# B&R Automation Studio project NAEUL004C00R13L518F00 (part 28)

#### Act_OptP1040Save.st
```iecst
ACTION Act_OptP1040Save:

	IF tyP1040ProdSet.tyProdSet.tyBtnSave.bRtCompl = TRUE THEN
		IF usiSaveProdRcpStep = 0 THEN
			//Mask Table
			tyP1040ProdSet.tyProdSet.tyStringSearch.uiMaskRtStat				:= FALSE;
			tyP1040ProdSet.tyProdSet.tyTableRecipe.uiMaskRtStat					:= FALSE;
			tyP1040ProdSet.tyProdSet.tyBtnDelete.uiMaskRtStat					:= FALSE;

			p_tyC0008MsgBox ACCESS ADR(tyP1040ProdSet.tyMsgBoxSaveAsk);

			IF tyP1040ProdSet.tyMsgBoxSaveAsk.tyBtnYes.bRtCompl = TRUE THEN
				tyP1040ProdSet.tyMsgBoxSaveAsk.tyBtnYes.bRtCompl				:= FALSE;
				tyP1040ProdSet.tyMsgBoxSaveAsk.tyBtnYes.bValue					:= FALSE;

				p_tyC0008MsgBox ACCESS ADR(tyP1040ProdSet.tyMsgBoxHide);

				usiSaveProdRcpStep	:= 1;

			ELSIF tyP1040ProdSet.tyMsgBoxSaveAsk.tyBtnNo.bRtCompl = TRUE THEN
				tyP1040ProdSet.tyMsgBoxSaveAsk.tyBtnNo.bRtCompl					:= FALSE;
				tyP1040ProdSet.tyMsgBoxSaveAsk.tyBtnNo.bValue					:= FALSE;

				p_tyC0008MsgBox ACCESS ADR(tyP1040ProdSet.tyMsgBoxHide);

				usiSaveProdRcpStep	:= 99;

			END_IF

		ELSIF usiSaveProdRcpStep = 1 THEN
			tyProdRcpInfoIn.sRcpNm				:= tyP1040ProdSet.tyProdSet.tyStringRecipeNm.sValue;
			tyProdRcpInfoIn.diWidthInUM			:= tyP1040ProdSet.tyProdSet.tyNumProdWidth.diValue;
			tyProdRcpInfoIn.diMaxSltValue		:= tyP1040ProdSet.tyProdSet.tyNumLastSlt.diValue;
			tyProdRcpInfoIn.diMinSltValue		:= tyP1040ProdSet.tyProdSet.tyNumFirstSlt.diValue;
			tyProdRcpInfoIn.diPitch				:= tyP1040ProdSet.tyProdSet.tyNumPitch.diValue;
			tyProdRcpInfoIn.diBrdPerSlt			:= tyP1040ProdSet.tyProdSet.tyNumBrdPerSlt.diValue;
			tyProdRcpInfoIn.usiMcMod			:= tyP1040ProdSet.tyProdSet.tyDrpDnMcMode.usiValueIdx;
			tyProdRcpInfoIn.bTopToBtm			:= tyP1040ProdSet.tyProdSet.tyBtnToptoBtm.bValue;
			tyProdRcpInfoIn.bGapBwtnBrd			:= tyP1040ProdSet.tyProdSet.tyBtnGapBetBrds.bValue;
			tyProdRcpInfoIn.bLongBrd			:= tyP1040ProdSet.tyProdSet.tyBtnLongBrd.bValue;
			tyProdRcpInfoIn.diMinReqFreeBffr	:= tyP1040ProdSet.tyProdSet.tyNumMinReqFreeBffr.diValue;
			tyProdRcpInfoIn.diMtrPshrExtSpd		:= tyP1040ProdSet.tyProdSet.tyNumMtrPshrExtSpd.diValue;
			tyProdRcpInfoIn.diMtrPshrExtTorq	:= tyP1040ProdSet.tyProdSet.tyNumMtrPshrExtTorq.diValue;
			tyProdRcpInfoIn.diPshrOffset		:= tyP1040ProdSet.tyProdSet.tyNumPshrOffset.diValue;

			IF p_tyNtParamCurr.bLFProdWidth2Prep THEN
				tyProdRcpInfoIn.diWidthInUM2		:= tyP1040ProdSet.tyProdSet.tyNumProdWidth2.diValue;// ADD
			ELSE
				tyProdRcpInfoIn.diWidthInUM2		:= tyP1040ProdSet.tyProdSet.tyNumProdWidth.diValue;// ADD
			END_IF

			eProdRcpAct	:= ProdRcpActAddEdit;

			IF p_eProdRcpStat = ProdRcpActAddEdit AND p_eProdRcpStatus = Done THEN
				eProdRcpAct	:= ProdRcpActIdle;

				IF p_bProdRcpNmEmpty = TRUE THEN
					usiSaveProdRcpStep		:= 2;
				ELSIF p_bProdRcpListFull = TRUE THEN
					usiSaveProdRcpStep		:= 3;
				ELSE
					tyP1040ProdSet.tyProdSet.tyBtnSort.bValue := FALSE;
					bRefreshProdRcpTable	:= TRUE;
					bRefreshProdRcpDetail	:= TRUE;
					usiSaveProdRcpStep		:= 4;
				END_IF

			ELSIF p_eProdRcpStatus = Error THEN
				p_tyC0008MsgBox ACCESS ADR(tyP1040ProdSet.tyMsgBoxSaveErr);

				IF tyP1040ProdSet.tyMsgBoxSaveErr.tyBtnNo.bRtCompl = TRUE THEN
					tyP1040ProdSet.tyMsgBoxSaveErr.tyBtnNo.bRtCompl 			:= FALSE;
					tyP1040ProdSet.tyMsgBoxSaveErr.tyBtnNo.bValue 				:= FALSE;

					p_tyC0008MsgBox ACCESS ADR(tyP1040ProdSet.tyMsgBoxHide);

					usiSaveProdRcpStep		:= 99;
				END_IF
			END_IF

		// Product Recipe Param Error
		ELSIF usiSaveProdRcpStep = 2 THEN
			p_tyC0008MsgBox ACCESS ADR(tyP1040ProdSet.tyMsgBoxSaveNoNm);

			IF tyP1040ProdSet.tyMsgBoxSaveNoNm.tyBtnNo.bRtCompl = TRUE THEN
				tyP1040ProdSet.tyMsgBoxSaveNoNm.tyBtnNo.bRtCompl 				:= FALSE;
				tyP1040ProdSet.tyMsgBoxSaveNoNm.tyBtnNo.bValue 					:= FALSE;

				p_tyC0008MsgBox ACCESS ADR(tyP1040ProdSet.tyMsgBoxHide);

				usiSaveProdRcpStep		:= 99;
			END_IF

		// Prod Recipe List Full
		ELSIF usiSaveProdRcpStep = 3 THEN
			p_tyC0008MsgBox ACCESS ADR(tyP1040ProdSet.tyMsgBoxListFull);

			IF tyP1040ProdSet.tyMsgBoxListFull.tyBtnNo.bRtCompl = TRUE THEN
				tyP1040ProdSet.tyMsgBoxListFull.tyBtnNo.bRtCompl 				:= FALSE;
				tyP1040ProdSet.tyMsgBoxListFull.tyBtnNo.bValue 					:= FALSE;

				p_tyC0008MsgBox ACCESS ADR(tyP1040ProdSet.tyMsgBoxHide);

				usiSaveProdRcpStep		:= 99;
			END_IF

		ELSIF usiSaveProdRcpStep = 4 THEN
			IF tyProdRcpInfoIn.sRcpNm = p_tyProdRcpCurrRcp0.sRcpNm THEN
				p_tyC0008MsgBox ACCESS ADR(tyP1040ProdSet.tyMsgBoxReloadCurrRcp);

				IF tyP1040ProdSet.tyMsgBoxReloadCurrRcp.tyBtnNo.bRtCompl = TRUE THEN
					tyP1040ProdSet.tyMsgBoxReloadCurrRcp.tyBtnNo.bRtCompl 		:= FALSE;
					tyP1040ProdSet.tyMsgBoxReloadCurrRcp.tyBtnNo.bValue 		:= FALSE;

					p_tyC0008MsgBox ACCESS ADR(tyP1040ProdSet.tyMsgBoxHide);

					usiSaveProdRcpStep		:= 99;
				END_IF
			ELSE
				usiSaveProdRcpStep			:= 99;
			END_IF

		ELSIF usiSaveProdRcpStep = 99 THEN
			bRefreshProdRcpTable 			:= FALSE;

			//Unmask
			tyP1040ProdSet.tyProdSet.tyStringSearch.uiMaskRtStat	:= TRUE;
			tyP1040ProdSet.tyProdSet.tyTableRecipe.uiMaskRtStat		:= TRUE;
			tyP1040ProdSet.tyProdSet.tyBtnDelete.uiMaskRtStat		:= TRUE;

			//Reset
			tyP1040ProdSet.tyProdSet.tyBtnSave.bRtCompl	:= FALSE;
			tyP1040ProdSet.tyProdSet.tyBtnSave.bValue	:= FALSE;

			usiSaveProdRcpStep	:= 0;

		END_IF

	END_IF

END_ACTION
```

#### Act_OptP1040LoadData.st
```iecst
ACTION Act_OptP1040LoadData:

	udiP1040SelectedRow		:= STRING_TO_UDINT(tyP1040ProdSet.tyProdSet.tyTableRecipe.a_tyStringDataCol0[tyP1040Table.uiSelectedRow].sValue);

	IF udiP1040SelectedRow <> udiP1040SelectedRowOld OR bRefreshProdRcpDetail = TRUE OR bUpdateP1040LoadData THEN
		IF tyP1040ProdSet.tyProdSet.tyStringSearch.sValue = '' THEN
			IF tyP1040ProdSet.tyProdSet.tyTableRecipe.a_tyStringDataCol1[tyP1040Table.uiSelectedRow].sValue <> '' THEN
				//Update Recipe Data
				IF tyP1040ProdSet.tyProdSet.tyBtnSort.bValue THEN
					tyP1040ProdSet.tyProdSet.tyStringRecipeNm.sValue		:= p_tyProdRcpSortedList[udiP1040SelectedRow].sRcpNm;
					tyP1040ProdSet.tyProdSet.tyNumProdWidth.diValue			:= p_tyProdRcpSortedList[udiP1040SelectedRow].diWidthInUM;
					tyP1040ProdSet.tyProdSet.tyNumProdWidth2.diValue		:= p_tyProdRcpSortedList[udiP1040SelectedRow].diWidthInUM2;
					tyP1040ProdSet.tyProdSet.tyNumLastSlt.diValue			:= p_tyProdRcpSortedList[udiP1040SelectedRow].diMaxSltValue;
					tyP1040ProdSet.tyProdSet.tyNumFirstSlt.diValue			:= p_tyProdRcpSortedList[udiP1040SelectedRow].diMinSltValue;
					tyP1040ProdSet.tyProdSet.tyNumPitch.diValue				:= p_tyProdRcpSortedList[udiP1040SelectedRow].diPitch;
					tyP1040ProdSet.tyProdSet.tyNumBrdPerSlt.diValue			:= p_tyProdRcpSortedList[udiP1040SelectedRow].diBrdPerSlt;
					tyP1040ProdSet.tyProdSet.tyDrpDnMcMode.usiValueIdx		:= p_tyProdRcpSortedList[udiP1040SelectedRow].usiMcMod;
					tyP1040ProdSet.tyProdSet.tyBtnToptoBtm.bValue			:= p_tyProdRcpSortedList[udiP1040SelectedRow].bTopToBtm;
					tyP1040ProdSet.tyProdSet.tyBtnGapBetBrds.bValue			:= p_tyProdRcpSortedList[udiP1040SelectedRow].bGapBwtnBrd;
					tyP1040ProdSet.tyProdSet.tyBtnLongBrd.bValue			:= p_tyProdRcpSortedList[udiP1040SelectedRow].bLongBrd;
					tyP1040ProdSet.tyProdSet.tyNumMinReqFreeBffr.diValue	:= p_tyProdRcpSortedList[udiP1040SelectedRow].diMinReqFreeBffr;
					tyP1040ProdSet.tyProdSet.tyNumMtrPshrExtSpd.diValue		:= p_tyProdRcpSortedList[udiP1040SelectedRow].diMtrPshrExtSpd;
					tyP1040ProdSet.tyProdSet.tyNumMtrPshrExtTorq.diValue	:= p_tyProdRcpSortedList[udiP1040SelectedRow].diMtrPshrExtTorq;
					tyP1040ProdSet.tyProdSet.tyNumPshrOffset.diValue		:= p_tyProdRcpSortedList[udiP1040SelectedRow].diPshrOffset;
				ELSE

					tyP1040ProdSet.tyProdSet.tyStringRecipeNm.sValue		:= p_tyProdRcpCurrList[udiP1040SelectedRow].sRcpNm;
					tyP1040ProdSet.tyProdSet.tyNumProdWidth.diValue			:= p_tyProdRcpCurrList[udiP1040SelectedRow].diWidthInUM;
					tyP1040ProdSet.tyProdSet.tyNumProdWidth2.diValue		:= p_tyProdRcpCurrList[udiP1040SelectedRow].diWidthInUM2;
					tyP1040ProdSet.tyProdSet.tyNumLastSlt.diValue			:= p_tyProdRcpCurrList[udiP1040SelectedRow].diMaxSltValue;
					tyP1040ProdSet.tyProdSet.tyNumFirstSlt.diValue			:= p_tyProdRcpCurrList[udiP1040SelectedRow].diMinSltValue;
					tyP1040ProdSet.tyProdSet.tyNumPitch.diValue				:= p_tyProdRcpCurrList[udiP1040SelectedRow].diPitch;
					tyP1040ProdSet.tyProdSet.tyNumBrdPerSlt.diValue			:= p_tyProdRcpCurrList[udiP1040SelectedRow].diBrdPerSlt;
					tyP1040ProdSet.tyProdSet.tyDrpDnMcMode.usiValueIdx		:= p_tyProdRcpCurrList[udiP1040SelectedRow].usiMcMod;
					tyP1040ProdSet.tyProdSet.tyBtnToptoBtm.bValue			:= p_tyProdRcpCurrList[udiP1040SelectedRow].bTopToBtm;
					tyP1040ProdSet.tyProdSet.tyBtnGapBetBrds.bValue			:= p_tyProdRcpCurrList[udiP1040SelectedRow].bGapBwtnBrd;
					tyP1040ProdSet.tyProdSet.tyBtnLongBrd.bValue			:= p_tyProdRcpCurrList[udiP1040SelectedRow].bLongBrd;
					tyP1040ProdSet.tyProdSet.tyNumMinReqFreeBffr.diValue	:= p_tyProdRcpCurrList[udiP1040SelectedRow].diMinReqFreeBffr;
					tyP1040ProdSet.tyProdSet.tyNumMtrPshrExtSpd.diValue		:= p_tyProdRcpCurrList[udiP1040SelectedRow].diMtrPshrExtSpd;
					tyP1040ProdSet.tyProdSet.tyNumMtrPshrExtTorq.diValue	:= p_tyProdRcpCurrList[udiP1040SelectedRow].diMtrPshrExtTorq;
					tyP1040ProdSet.tyProdSet.tyNumPshrOffset.diValue		:= p_tyProdRcpCurrList[udiP1040SelectedRow].diPshrOffset;
				END_IF
			ELSE
				tyP1040ProdSet.tyProdSet.tyStringRecipeNm.sValue		:= '';
				tyP1040ProdSet.tyProdSet.tyNumProdWidth.diValue			:= 100000;
				tyP1040ProdSet.tyProdSet.tyNumProdWidth2.diValue		:= 100000;
				tyP1040ProdSet.tyProdSet.tyNumLastSlt.diValue			:= p_tyMagRcpCurrRcp.diTtlSlt;
				tyP1040ProdSet.tyProdSet.tyNumFirstSlt.diValue			:= p_tyNtParamCurr.diProjMagMinSlt;
				tyP1040ProdSet.tyProdSet.tyNumPitch.diValue				:= 1;
				tyP1040ProdSet.tyProdSet.tyNumBrdPerSlt.diValue			:= 1;
				tyP1040ProdSet.tyProdSet.tyDrpDnMcMode.usiValueIdx		:= p_tyMcParamCurr.usiDefaultMcMod;
				tyP1040ProdSet.tyProdSet.tyBtnToptoBtm.bValue			:= FALSE;
				tyP1040ProdSet.tyProdSet.tyBtnGapBetBrds.bValue			:= FALSE;
				tyP1040ProdSet.tyProdSet.tyBtnLongBrd.bValue			:= FALSE;
				tyP1040ProdSet.tyProdSet.tyNumMinReqFreeBffr.diValue	:= 0;
				tyP1040ProdSet.tyProdSet.tyNumMtrPshrExtSpd.diValue		:= 8;
				tyP1040ProdSet.tyProdSet.tyNumMtrPshrExtTorq.diValue	:= 80;
				tyP1040ProdSet.tyProdSet.tyNumPshrOffset.diValue		:= 0;
			END_IF

		ELSE

			IF tyP1040ProdSet.tyProdSet.tyTableRecipe.a_tyStringDataCol1[tyP1040Table.uiSelectedRow].sValue <> '' THEN
				//Update Recipe Data
				IF tyP1040ProdSet.tyProdSet.tyBtnSort.bValue THEN
					tyP1040ProdSet.tyProdSet.tyStringRecipeNm.sValue		:= p_tyProdRcpSortedList[udiP1040SelectedRow].sRcpNm;
					tyP1040ProdSet.tyProdSet.tyNumProdWidth.diValue			:= p_tyProdRcpSortedList[udiP1040SelectedRow].diWidthInUM;
					tyP1040ProdSet.tyProdSet.tyNumProdWidth2.diValue		:= p_tyProdRcpSortedList[udiP1040SelectedRow].diWidthInUM2;
					tyP1040ProdSet.tyProdSet.tyNumLastSlt.diValue			:= p_tyProdRcpSortedList[udiP1040SelectedRow].diMaxSltValue;
					tyP1040ProdSet.tyProdSet.tyNumFirstSlt.diValue			:= p_tyProdRcpSortedList[udiP1040SelectedRow].diMinSltValue;
					tyP1040ProdSet.tyProdSet.tyNumPitch.diValue				:= p_tyProdRcpSortedList[udiP1040SelectedRow].diPitch;
					tyP1040ProdSet.tyProdSet.tyNumBrdPerSlt.diValue			:= p_tyProdRcpSortedList[udiP1040SelectedRow].diBrdPerSlt;
					tyP1040ProdSet.tyProdSet.tyDrpDnMcMode.usiValueIdx		:= p_tyProdRcpSortedList[udiP1040SelectedRow].usiMcMod;
					tyP1040ProdSet.tyProdSet.tyBtnToptoBtm.bValue			:= p_tyProdRcpSortedList[udiP1040SelectedRow].bTopToBtm;
					tyP1040ProdSet.tyProdSet.tyBtnGapBetBrds.bValue			:= p_tyProdRcpSortedList[udiP1040SelectedRow].bGapBwtnBrd;
					tyP1040ProdSet.tyProdSet.tyBtnLongBrd.bValue			:= p_tyProdRcpSortedList[udiP1040SelectedRow].bLongBrd;
					tyP1040ProdSet.tyProdSet.tyNumMinReqFreeBffr.diValue	:= p_tyProdRcpSortedList[udiP1040SelectedRow].diMinReqFreeBffr;
					tyP1040ProdSet.tyProdSet.tyNumMtrPshrExtSpd.diValue		:= p_tyProdRcpSortedList[udiP1040SelectedRow].diMtrPshrExtSpd;
					tyP1040ProdSet.tyProdSet.tyNumMtrPshrExtTorq.diValue	:= p_tyProdRcpSortedList[udiP1040SelectedRow].diMtrPshrExtTorq;
					tyP1040ProdSet.tyProdSet.tyNumPshrOffset.diValue		:= p_tyProdRcpSortedList[udiP1040SelectedRow].diPshrOffset;
				ELSE
					tyP1040ProdSet.tyProdSet.tyStringRecipeNm.sValue		:= p_tyProdRcpFilterList[udiP1040SelectedRow].sRcpNm;
					tyP1040ProdSet.tyProdSet.tyNumProdWidth.diValue			:= p_tyProdRcpFilterList[udiP1040SelectedRow].diWidthInUM;
					tyP1040ProdSet.tyProdSet.tyNumProdWidth2.diValue		:= p_tyProdRcpSortedList[udiP1040SelectedRow].diWidthInUM2;
					tyP1040ProdSet.tyProdSet.tyNumLastSlt.diValue			:= p_tyProdRcpFilterList[udiP1040SelectedRow].diMaxSltValue;
					tyP1040ProdSet.tyProdSet.tyNumFirstSlt.diValue			:= p_tyProdRcpFilterList[udiP1040SelectedRow].diMinSltValue;
					tyP1040ProdSet.tyProdSet.tyNumPitch.diValue				:= p_tyProdRcpFilterList[udiP1040SelectedRow].diPitch;
					tyP1040ProdSet.tyProdSet.tyNumBrdPerSlt.diValue			:= p_tyProdRcpFilterList[udiP1040SelectedRow].diBrdPerSlt;
					tyP1040ProdSet.tyProdSet.tyDrpDnMcMode.usiValueIdx		:= p_tyProdRcpFilterList[udiP1040SelectedRow].usiMcMod;
					tyP1040ProdSet.tyProdSet.tyBtnToptoBtm.bValue			:= p_tyProdRcpFilterList[udiP1040SelectedRow].bTopToBtm;
					tyP1040ProdSet.tyProdSet.tyBtnGapBetBrds.bValue			:= p_tyProdRcpFilterList[udiP1040SelectedRow].bGapBwtnBrd;
					tyP1040ProdSet.tyProdSet.tyBtnLongBrd.bValue			:= p_tyProdRcpFilterList[udiP1040SelectedRow].bLongBrd;
					tyP1040ProdSet.tyProdSet.tyNumMinReqFreeBffr.diValue	:= p_tyProdRcpFilterList[udiP1040SelectedRow].diMinReqFreeBffr;
					tyP1040ProdSet.tyProdSet.tyNumMtrPshrExtSpd.diValue		:= p_tyProdRcpFilterList[udiP1040SelectedRow].diMtrPshrExtSpd;
					tyP1040ProdSet.tyProdSet.tyNumMtrPshrExtTorq.diValue	:= p_tyProdRcpFilterList[udiP1040SelectedRow].diMtrPshrExtTorq;
					tyP1040ProdSet.tyProdSet.tyNumPshrOffset.diValue		:= p_tyProdRcpFilterList[udiP1040SelectedRow].diPshrOffset;
				END_IF
			ELSE
				tyP1040ProdSet.tyProdSet.tyStringRecipeNm.sValue		:= '';
				tyP1040ProdSet.tyProdSet.tyNumProdWidth.diValue			:= 100000;
				tyP1040ProdSet.tyProdSet.tyNumProdWidth2.diValue		:= 100000;
				tyP1040ProdSet.tyProdSet.tyNumLastSlt.diValue			:= p_tyMagRcpCurrRcp.diTtlSlt;
				tyP1040ProdSet.tyProdSet.tyNumFirstSlt.diValue			:= p_tyNtParamCurr.diProjMagMinSlt;
				tyP1040ProdSet.tyProdSet.tyNumPitch.diValue				:= 1;
				tyP1040ProdSet.tyProdSet.tyNumBrdPerSlt.diValue			:= 1;
				tyP1040ProdSet.tyProdSet.tyDrpDnMcMode.usiValueIdx		:= p_tyMcParamCurr.usiDefaultMcMod;
				tyP1040ProdSet.tyProdSet.tyBtnToptoBtm.bValue			:= FALSE;
				tyP1040ProdSet.tyProdSet.tyBtnGapBetBrds.bValue			:= FALSE;
				tyP1040ProdSet.tyProdSet.tyBtnLongBrd.bValue			:= FALSE;
				tyP1040ProdSet.tyProdSet.tyNumMinReqFreeBffr.diValue	:= 0;
				tyP1040ProdSet.tyProdSet.tyNumMtrPshrExtSpd.diValue		:= 8;
				tyP1040ProdSet.tyProdSet.tyNumMtrPshrExtTorq.diValue	:= 80;
				tyP1040ProdSet.tyProdSet.tyNumPshrOffset.diValue		:= 0;
			END_IF

		END_IF

		bUpdateP1040LoadData 		:= FALSE;
		bRefreshProdRcpDetail		:= FALSE;
		udiP1040SelectedRowOld 		:= udiP1040SelectedRow;

		fUIInRtStatOff(ADR(tyP1040ProdSet.tyProdSet.tyBtnSave.uiMaskRtStat));

	END_IF

END_ACTION
```

#### Act_OptP1040Del.st
```iecst
ACTION Act_OptP1040Del:

	IF tyP1040ProdSet.tyProdSet.tyBtnDelete.bRtCompl = TRUE THEN
		IF usiDelProdRcpStep = 0 THEN
			tyP1040ProdSet.tyProdSet.tyStringSearch.uiMaskRtStat				:= FALSE;
			tyP1040ProdSet.tyProdSet.tyTableRecipe.uiMaskRtStat					:= FALSE;

			IF tyP1040ProdSet.tyProdSet.tyTableRecipe.a_tyStringDataCol1[tyP1040Table.uiSelectedRow].sValue = p_tyProdRcpCurrRcp0.sRcpNm THEN
				p_tyC0008MsgBox ACCESS ADR(tyP1040ProdSet.tyMsgBoxDelCurrRcpAsk);

				IF tyP1040ProdSet.tyMsgBoxDelCurrRcpAsk.tyBtnNo.bRtCompl = TRUE THEN
					tyP1040ProdSet.tyMsgBoxDelCurrRcpAsk.tyBtnNo.bRtCompl 		:= FALSE;
					tyP1040ProdSet.tyMsgBoxDelCurrRcpAsk.tyBtnNo.bValue 		:= FALSE;

					p_tyC0008MsgBox ACCESS ADR(tyP1040ProdSet.tyMsgBoxHide);

					usiDelProdRcpStep	:= 99;
				END_IF
			ELSE
				p_tyC0008MsgBox ACCESS ADR(tyP1040ProdSet.tyMsgBoxDelAsk);

				IF tyP1040ProdSet.tyMsgBoxDelAsk.tyBtnYes.bRtCompl = TRUE THEN
					tyP1040ProdSet.tyMsgBoxDelAsk.tyBtnYes.bRtCompl				:= FALSE;
					tyP1040ProdSet.tyMsgBoxDelAsk.tyBtnYes.bValue				:= FALSE;

					p_tyC0008MsgBox ACCESS ADR(tyP1040ProdSet.tyMsgBoxHide);

					usiDelProdRcpStep	:= 1;

				ELSIF tyP1040ProdSet.tyMsgBoxDelAsk.tyBtnNo.bRtCompl = TRUE THEN
					tyP1040ProdSet.tyMsgBoxDelAsk.tyBtnNo.bRtCompl				:= FALSE;
					tyP1040ProdSet.tyMsgBoxDelAsk.tyBtnNo.bValue				:= FALSE;

					p_tyC0008MsgBox ACCESS ADR(tyP1040ProdSet.tyMsgBoxHide);

					usiDelProdRcpStep	:= 99;

				END_IF
			END_IF

		ELSIF usiDelProdRcpStep = 1 THEN
			tyProdRcpInfoIn.sRcpNm			:= tyP1040ProdSet.tyProdSet.tyTableRecipe.a_tyStringDataCol1[tyP1040Table.uiSelectedRow].sValue;

			eProdRcpAct					:= ProdRcpActDel;

			IF p_eProdRcpStat = ProdRcpActDel AND p_eProdRcpStatus = Done THEN
				eProdRcpAct				:= ProdRcpActIdle;

				IF p_bProdRcpNmEmpty = TRUE THEN
					usiDelProdRcpStep		:= 2;
				ELSIF p_bProdRcpNmNotExist = TRUE THEN
					usiDelProdRcpStep		:= 3;
				ELSE
					tyP1040ProdSet.tyProdSet.tyBtnSort.bValue := FALSE;
					bRefreshProdRcpTable	:= TRUE;
					bRefreshProdRcpDetail	:= TRUE;
					usiDelProdRcpStep		:= 99;
				END_IF

			ELSIF p_eProdRcpStatus = Error THEN
				p_tyC0008MsgBox ACCESS ADR(tyP1040ProdSet.tyMsgBoxDelErr);

				IF tyP1040ProdSet.tyMsgBoxDelErr.tyBtnNo.bRtCompl = TRUE THEN
					tyP1040ProdSet.tyMsgBoxDelErr.tyBtnNo.bRtCompl 				:= FALSE;
					tyP1040ProdSet.tyMsgBoxDelErr.tyBtnNo.bValue 				:= FALSE;

					p_tyC0008MsgBox ACCESS ADR(tyP1040ProdSet.tyMsgBoxHide);

					usiDelProdRcpStep		:= 99;
				END_IF
			END_IF

		ELSIF usiDelProdRcpStep = 2 THEN
			p_tyC0008MsgBox ACCESS ADR(tyP1040ProdSet.tyMsgBoxDelNmEmpty);

			IF tyP1040ProdSet.tyMsgBoxDelNmEmpty.tyBtnNo.bRtCompl = TRUE THEN
				tyP1040ProdSet.tyMsgBoxDelNmEmpty.tyBtnNo.bRtCompl 				:= FALSE;
				tyP1040ProdSet.tyMsgBoxDelNmEmpty.tyBtnNo.bValue 				:= FALSE;

				p_tyC0008MsgBox ACCESS ADR(tyP1040ProdSet.tyMsgBoxHide);

				usiDelProdRcpStep		:= 99;
			END_IF

		ELSIF usiDelProdRcpStep = 3 THEN
			p_tyC0008MsgBox ACCESS ADR(tyP1040ProdSet.tyMsgBoxDelNmNotExist);

			IF tyP1040ProdSet.tyMsgBoxDelNmNotExist.tyBtnNo.bRtCompl = TRUE THEN
				tyP1040ProdSet.tyMsgBoxDelNmNotExist.tyBtnNo.bRtCompl 		:= FALSE;
				tyP1040ProdSet.tyMsgBoxDelNmNotExist.tyBtnNo.bValue 		:= FALSE;

				p_tyC0008MsgBox ACCESS ADR(tyP1040ProdSet.tyMsgBoxHide);

				usiDelProdRcpStep	:= 99;
			END_IF

		ELSIF usiDelProdRcpStep = 99 THEN
			bRefreshProdRcpTable	:= FALSE;

			//Unmask
			tyP1040ProdSet.tyProdSet.tyStringSearch.uiMaskRtStat			:= TRUE;
			tyP1040ProdSet.tyProdSet.tyTableRecipe.uiMaskRtStat				:= TRUE;

			//Reset
			tyP1040ProdSet.tyProdSet.tyBtnDelete.bRtCompl					:= FALSE;
			tyP1040ProdSet.tyProdSet.tyBtnDelete.bValue						:= FALSE;

			usiDelProdRcpStep		:= 0;
		END_IF

	END_IF

END_ACTION
```

#### Act_OptP1040Table.st
```iecst
ACTION Act_OptP1040Table:

	//Call Table FB
	fbP1040Table.sVisuNm			:= tyP1040Table.sVisuNm;
	fbP1040Table.udiWorkAreaStartX	:= 359;
	fbP1040Table.udiWorkAreaEndX	:= 770;
	fbP1040Table.udiWorkAreaStartY	:= 93;
	fbP1040Table.udiWorkAreaEndY	:= 415;
	fbP1040Table.udiMinXDist		:= 20;
	fbP1040Table.udiMinYDist		:= 20;
	fbP1040Table.uiSlideScale		:= c_uiP1040TableSize;
	fbP1040Table.iTotalData			:= UDINT_TO_INT(c_udiProdRcpMax);
	fbP1040Table.iTotalRow			:= c_uiP1040TableSize;
	fbP1040Table.p_uiSliderStatus	:= ADR(tyP1040ProdSet.tyProdSet.tyTableRecipe.tyUISlider.uiRtStat);
	fbP1040Table.pa_tyUIHotspot		:= ADR(tyP1040ProdSet.tyProdSet.tyTableRecipe.a_tyHotspot);
	fbP1040Table.p_uiTablePos		:= ADR(tyP1040Table.uiTablePos);
	fbP1040Table.p_iSliderPos		:= ADR(tyP1040ProdSet.tyProdSet.tyTableRecipe.tyUISlider.iValue);
	fbP1040Table.p_uiSelectedRow	:= ADR(tyP1040Table.uiSelectedRow);
	fbP1040Table.p_bTableActive		:= ADR(tyP1040Table.bTableActive);
	fbP1040Table.p_bSliderActive	:= ADR(tyP1040Table.bSliderActive);
	fbP1040Table;

	//Table Content
	IF tyP1040Table.bTableActive = TRUE OR tyP1040Table.bSliderActive = TRUE OR bRefreshProdRcpTable = TRUE OR bUpdateP1040Table THEN
		FOR i := 1 TO c_uiP1040TableSize DO
			IF tyP1040ProdSet.tyProdSet.tyBtnSort.bValue THEN
				tyP1040ProdSet.tyProdSet.tyTableRecipe.a_tyStringDataCol0[i].sValue	    := UINT_TO_STRING(tyP1040Table.uiTablePos + i - 1);
				tyP1040ProdSet.tyProdSet.tyTableRecipe.a_tyStringDataCol1[i].sValue		:= p_tyProdRcpSortedList[tyP1040Table.uiTablePos + i - 1].sRcpNm;
				tyP1040ProdSet.tyProdSet.tyTableRecipe.a_tyStringDataCol2[i].sValue		:= p_tyProdRcpSortedList[tyP1040Table.uiTablePos + i - 1].sDisplayInfo;
			ELSE

				IF tyP1040ProdSet.tyProdSet.tyStringSearch.sValue = '' THEN
					tyP1040ProdSet.tyProdSet.tyTableRecipe.a_tyStringDataCol0[i].sValue	    := UINT_TO_STRING(tyP1040Table.uiTablePos + i - 1);
					tyP1040ProdSet.tyProdSet.tyTableRecipe.a_tyStringDataCol1[i].sValue		:= p_tyProdRcpCurrList[tyP1040Table.uiTablePos + i - 1].sRcpNm;
					tyP1040ProdSet.tyProdSet.tyTableRecipe.a_tyStringDataCol2[i].sValue		:= p_tyProdRcpCurrList[tyP1040Table.uiTablePos + i - 1].sDisplayInfo;
				ELSE
					tyP1040ProdSet.tyProdSet.tyTableRecipe.a_tyStringDataCol0[i].sValue		:= UINT_TO_STRING(tyP1040Table.uiTablePos + i - 1);
					tyP1040ProdSet.tyProdSet.tyTableRecipe.a_tyStringDataCol1[i].sValue		:= p_tyProdRcpFilterList[tyP1040Table.uiTablePos + i - 1].sRcpNm;
					tyP1040ProdSet.tyProdSet.tyTableRecipe.a_tyStringDataCol2[i].sValue		:= p_tyProdRcpFilterList[tyP1040Table.uiTablePos + i - 1].sDisplayInfo;
				END_IF
			END_IF

		END_FOR

		IF bUpdateP1040Table THEN
			bUpdateP1040Table := FALSE;
		END_IF
	END_IF

	//Selected Row
	IF tyP1040Table.uiSelectedRow <> tyP1040Table.uiSelectedRowOld THEN
		FOR i := 1 TO c_uiP1040TableSize DO
			IF tyP1040Table.uiSelectedRow = i THEN
				tyP1040ProdSet.tyProdSet.tyTableRecipe.a_tyStringDataCol1[i].usiColor	:= 1;
				tyP1040ProdSet.tyProdSet.tyTableRecipe.a_tyStringDataCol2[i].usiColor	:= 1;
			ELSE
				tyP1040ProdSet.tyProdSet.tyTableRecipe.a_tyStringDataCol1[i].usiColor	:= 0;
				tyP1040ProdSet.tyProdSet.tyTableRecipe.a_tyStringDataCol2[i].usiColor	:= 0;
			END_IF
		END_FOR

		tyP1040Table.uiSelectedRowOld	:= tyP1040Table.uiSelectedRow;
	END_IF

END_ACTION
```

#### Act_OptP1040Search.st
```iecst
ACTION Act_OptP1040Search:

	IF tyP1040ProdSet.tyProdSet.tyStringSearch.bRtCompl = TRUE THEN	//Search Input Valid
		IF tyP1040ProdSet.tyProdSet.tyStringSearch.sValue = '' THEN
			FOR i := 1 TO c_uiP1040TableSize DO
				tyP1040ProdSet.tyProdSet.tyTableRecipe.a_tyStringDataCol0[i].sValue			:= UINT_TO_STRING(tyP1040Table.uiTablePos + i - 1);
				tyP1040ProdSet.tyProdSet.tyTableRecipe.a_tyStringDataCol1[i].sValue			:= p_tyProdRcpCurrList[tyP1040Table.uiTablePos + i - 1].sRcpNm;
				tyP1040ProdSet.tyProdSet.tyTableRecipe.a_tyStringDataCol2[i].sValue			:= p_tyProdRcpCurrList[tyP1040Table.uiTablePos + i - 1].sDisplayInfo;
			END_FOR

			tyP1040ProdSet.tyProdSet.tyStringSearch.bRtCompl			:= FALSE;
			bRefreshProdRcpDetail										:= TRUE;

			IF tyP1040ProdSet.tyProdSet.tyBtnSort.bValue THEN
				bFilterSortP1040	:= TRUE;
			END_IF

		ELSE
			tyP1040ProdSet.tyProdSet.tyTableRecipe.uiMaskRtStat			:= FALSE;
			tyP1040ProdSet.tyProdSet.tyBtnSave.uiMaskRtStat				:= FALSE;
			tyP1040ProdSet.tyProdSet.tyBtnDelete.uiMaskRtStat			:= FALSE;

			sProdRcpSearch			:= tyP1040ProdSet.tyProdSet.tyStringSearch.sValue;

			eProdRcpAct			:= ProdRcpActFilter;

			IF p_eProdRcpStat = ProdRcpActFilter AND p_eProdRcpStatus = Done THEN
				eProdRcpAct		:= ProdRcpActIdle;

				FOR i := 1 TO c_uiP1040TableSize DO
					tyP1040ProdSet.tyProdSet.tyTableRecipe.a_tyStringDataCol0[i].sValue		:= UINT_TO_STRING(tyP1040Table.uiTablePos + i - 1);
					tyP1040ProdSet.tyProdSet.tyTableRecipe.a_tyStringDataCol1[i].sValue		:= p_tyProdRcpFilterList[tyP1040Table.uiTablePos + i - 1].sRcpNm;
					tyP1040ProdSet.tyProdSet.tyTableRecipe.a_tyStringDataCol2[i].sValue		:= p_tyProdRcpFilterList[tyP1040Table.uiTablePos + i - 1].sDisplayInfo;
				END_FOR

				//Unmask Table
				tyP1040ProdSet.tyProdSet.tyTableRecipe.uiMaskRtStat		:= TRUE;
				tyP1040ProdSet.tyProdSet.tyBtnSave.uiMaskRtStat			:= FALSE;
				tyP1040ProdSet.tyProdSet.tyBtnDelete.uiMaskRtStat		:= TRUE;

				//Reset
				tyP1040ProdSet.tyProdSet.tyStringSearch.bRtCompl		:= FALSE;
				bRefreshProdRcpDetail									:= TRUE;

				IF tyP1040ProdSet.tyProdSet.tyBtnSort.bValue THEN
					bFilterSortP1040	:= TRUE;
				END_IF

			ELSIF p_eProdRcpStatus = Error THEN
				FOR i := 1 TO c_uiP1040TableSize DO
					tyP1040ProdSet.tyProdSet.tyTableRecipe.a_tyStringDataCol0[i].sValue		:= UINT_TO_STRING(tyP1040Table.uiTablePos + i - 1);
					tyP1040ProdSet.tyProdSet.tyTableRecipe.a_tyStringDataCol1[i].sValue		:= '';
					tyP1040ProdSet.tyProdSet.tyTableRecipe.a_tyStringDataCol2[i].sValue		:= '';
				END_FOR

				p_tyC0008MsgBox ACCESS ADR (tyP1040ProdSet.tyMsgBoxListErr);

				IF tyP1040ProdSet.tyMsgBoxListErr.tyBtnNo.bRtCompl = TRUE THEN
					tyP1040ProdSet.tyMsgBoxListErr.tyBtnNo.bRtCompl 	:= TRUE;
					tyP1040ProdSet.tyMsgBoxListErr.tyBtnNo.bValue		:= TRUE;

					p_tyC0008MsgBox ACCESS ADR (tyP1040ProdSet.tyMsgBoxHide);

					//Unmask Table
					tyP1040ProdSet.tyProdSet.tyTableRecipe.uiMaskRtStat	:= TRUE;
					tyP1040ProdSet.tyProdSet.tyBtnSave.uiMaskRtStat		:= FALSE;
					tyP1040ProdSet.tyProdSet.tyBtnDelete.uiMaskRtStat	:= TRUE;

					//Reset
					tyP1040ProdSet.tyProdSet.tyStringSearch.bRtCompl	:= FALSE;
					bRefreshProdRcpDetail								:= TRUE;
				END_IF
			END_IF
		END_IF
	END_IF

END_ACTION
```

#### Act_OptP1040Keypad.st
```iecst
ACTION Act_OptP1040Keypad:

	tyP1040ProdSet.tyProdSet.tyNumFirstSlt.diValueMax	:= tyP1040ProdSet.tyProdSet.tyNumLastSlt.diValue;
	tyP1040ProdSet.tyProdSet.tyNumLastSlt.diValueMin	:= tyP1040ProdSet.tyProdSet.tyNumFirstSlt.diValue;
	tyP1040ProdSet.tyProdSet.tyNumPitch.diValueMax		:= tyP1040ProdSet.tyProdSet.tyNumLastSlt.diValue - tyP1040ProdSet.tyProdSet.tyNumFirstSlt.diValue + 1;

	IF fUIOutRtStatTPIsOpen(ADR(tyP1040ProdSet.tyProdSet.tyStringRecipeNm.uiRtStat)) THEN
		tyProperty.tyKeypad.tyStringTitle.sKeypadTitle	:= tyP1040ProdSet.tyProdSet.tyStringRecipeNm.sKeypadTitle;

	ELSIF fUIOutRtStatTPIsOpen(ADR(tyP1040ProdSet.tyProdSet.tyNumProdWidth.uiRtStat)) THEN
		IF p_tyNtParamCurr.bLFProdWidth2Prep THEN
			tyProperty.tyKeypad.tyTxtTitle.sTxt	:= 'Product Width US';
		ELSE
			tyProperty.tyKeypad.tyTxtTitle.sTxt	:= 'Product Width';
		END_IF

	ELSIF fUIOutRtStatTPIsOpen(ADR(tyP1040ProdSet.tyProdSet.tyNumProdWidth2.uiRtStat)) THEN
		tyProperty.tyKeypad.tyTxtTitle.sTxt	:='Product Width DS';

	ELSIF fUIOutRtStatTPIsOpen(ADR(tyP1040ProdSet.tyProdSet.tyStringSearch.uiRtStat)) THEN
		tyProperty.tyKeypad.tyStringTitle.sKeypadTitle	:= tyP1040ProdSet.tyProdSet.tyStringSearch.sKeypadTitle;

	ELSIF fUIOutRtStatTPIsOpen(ADR(tyP1040ProdSet.tyProdSet.tyNumFirstSlt.uiRtStat)) THEN
		tyProperty.tyKeypad.tyStringTitle.sKeypadTitle	:= tyP1040ProdSet.tyProdSet.tyNumFirstSlt.sKeypadTitle;

	ELSIF fUIOutRtStatTPIsOpen(ADR(tyP1040ProdSet.tyProdSet.tyNumLastSlt.uiRtStat)) THEN
		tyProperty.tyKeypad.tyStringTitle.sKeypadTitle	:= tyP1040ProdSet.tyProdSet.tyNumLastSlt.sKeypadTitle;

	ELSIF fUIOutRtStatTPIsOpen(ADR(tyP1040ProdSet.tyProdSet.tyNumPitch.uiRtStat)) THEN
		tyProperty.tyKeypad.tyStringTitle.sKeypadTitle	:= tyP1040ProdSet.tyProdSet.tyNumPitch.sKeypadTitle;

	ELSIF fUIOutRtStatTPIsOpen(ADR(tyP1040ProdSet.tyProdSet.tyNumMinReqFreeBffr.uiRtStat)) THEN
		tyProperty.tyKeypad.tyStringTitle.sKeypadTitle	:= tyP1040ProdSet.tyProdSet.tyNumMinReqFreeBffr.sKeypadTitle;

	ELSIF fUIOutRtStatTPIsOpen(ADR(tyP1040ProdSet.tyProdSet.tyNumBrdPerSlt.uiRtStat)) THEN
		tyProperty.tyKeypad.tyStringTitle.sKeypadTitle	:= tyP1040ProdSet.tyProdSet.tyNumBrdPerSlt.sKeypadTitle;

	ELSIF fUIOutRtStatTPIsOpen(ADR(tyP1040ProdSet.tyProdSet.tyNumPshrOffset.uiRtStat))THEN
		tyProperty.tyKeypad.tyStringTitle.sKeypadTitle	:= tyP1040ProdSet.tyProdSet.tyNumPshrOffset.sKeypadTitle;

	ELSE
		tyProperty.tyKeypad.tyStringTitle.sKeypadTitle	:= '';

	END_IF

END_ACTION
```

#### Act_OptP1040Limit.st
```iecst
ACTION Act_OptP1040Limit:

//	IF tyP1040ProdSet.tyProdSet.tyTableRecipe.a_tyStringDataCol1[udiP1040SelectedRow].sValue <> '' THEN
//		tyP1040ProdSet.tyProdSet.tyNumPshrOffset.diValueMin		:= -(p_tyProdRcpCurrList[udiP1040SelectedRow].diWidthInUM/2-p_tyMcParamCurr.diAWPusherAtHmPosInUM-5000);
//		tyP1040ProdSet.tyProdSet.tyNumPshrOffset.diValueMax		:= (p_tyProdRcpCurrList[udiP1040SelectedRow].diWidthInUM/2-p_tyMcParamCurr.diAWPusherAtHmPosInUM-5000);
//	ELSE
//		tyP1040ProdSet.tyProdSet.tyNumPshrOffset.diValueMin		:= 0;
//		tyP1040ProdSet.tyProdSet.tyNumPshrOffset.diValueMax		:= 0;
//	END_IF

	//Pusher Offset has to include min safe zone and max safe zone for the product width // 04102022 - 2022-0617
	IF (tyP1040ProdSet.tyProdSet.tyNumProdWidth.diValue) <> 0 THEN
		tyP1040ProdSet.tyProdSet.tyNumPshrOffset.diValueMin	:= - ((tyP1040ProdSet.tyProdSet.tyNumProdWidth.diValue/2 - p_tyMcParamCurr.diAWPusherAtHmPosInUM) - IPshrSafeDistanceValue);
		tyP1040ProdSet.tyProdSet.tyNumPshrOffset.diValueMax	:= ((tyP1040ProdSet.tyProdSet.tyNumProdWidth.diValue/2 - p_tyMcParamCurr.diAWPusherAtHmPosInUM) - IPshrSafeDistanceValue);
	ELSE
		tyP1040ProdSet.tyProdSet.tyNumPshrOffset.diValueMin	:= 0;
		tyP1040ProdSet.tyProdSet.tyNumPshrOffset.diValueMax	:= 0;
	END_IF

END_ACTION
```

#### Act_OptP1040Sort.st
```iecst
ACTION Act_OptP1040Sort:

	IF tyP1040ProdSet.tyProdSet.tyBtnSort.bValue THEN
		tyP1040ProdSet.tyProdSet.tyBtnSort.usiTxtIdx 	:= 1;
	ELSE
		tyP1040ProdSet.tyProdSet.tyBtnSort.usiTxtIdx 	:= 0;
	END_IF

	IF tyP1040ProdSet.tyProdSet.tyBtnSort.bRtCompl THEN
		bUpdateP1040LoadData := TRUE;
	END_IF

	IF tyP1040ProdSet.tyProdSet.tyBtnSort.bRtCompl OR (bFilterSortP1040 AND p_eProdRcpStat<> ProdRcpActFilter) THEN

		IF tyP1040ProdSet.tyProdSet.tyBtnSort.bValue THEN

			tyP1040ProdSet.tyProdSet.tyTableRecipe.uiMaskRtStat.0	:= FALSE;

			sProdRcpSearch	:= tyP1040ProdSet.tyProdSet.tyStringSearch.sValue;

			eProdRcpAct	:= ProdRcpActSort;

			IF p_eProdRcpStat = ProdRcpActSort AND p_eProdRcpStatus = Done THEN
				eProdRcpAct		:= ProdRcpActIdle;

				FOR i := 1 TO c_uiP1040TableSize DO
					tyP1040ProdSet.tyProdSet.tyTableRecipe.a_tyStringDataCol0[i].sValue	:= UINT_TO_STRING(tyP1040Table.uiTablePos + i - 1);
					tyP1040ProdSet.tyProdSet.tyTableRecipe.a_tyStringDataCol1[i].sValue	:= p_tyProdRcpSortedList[tyP1040Table.uiTablePos + i - 1].sRcpNm;
					tyP1040ProdSet.tyProdSet.tyTableRecipe.a_tyStringDataCol2[i].sValue	:= p_tyProdRcpSortedList[tyP1040Table.uiTablePos + i - 1].sDisplayInfo;
				END_FOR

				bFilterSortP1040	:= FALSE;

				//Unmask
				tyP1040ProdSet.tyProdSet.tyTableRecipe.uiMaskRtStat.0	:= TRUE;

				tyP1040ProdSet.tyProdSet.tyBtnSort.bRtCompl := FALSE;

			ELSIF p_eProdRcpStatus = Error THEN
				FOR i := 1 TO c_uiP1040TableSize DO
					tyP1040ProdSet.tyProdSet.tyTableRecipe.a_tyStringDataCol0[i].sValue		:= UINT_TO_STRING(tyP1040Table.uiTablePos + i - 1);
					tyP1040ProdSet.tyProdSet.tyTableRecipe.a_tyStringDataCol1[i].sValue		:= '';
					tyP1040ProdSet.tyProdSet.tyTableRecipe.a_tyStringDataCol2[i].sValue		:= '';
				END_FOR

				p_tyC0008MsgBox ACCESS ADR (tyP1040ProdSet.tyMsgBoxListErr);

				bFilterSortP1040	:= FALSE;

				IF tyP1040ProdSet.tyMsgBoxListErr.tyBtnNo.bRtCompl = TRUE THEN
					tyP1040ProdSet.tyMsgBoxListErr.tyBtnNo.bRtCompl 		:= TRUE;
					tyP1040ProdSet.tyMsgBoxListErr.tyBtnNo.bValue			:= TRUE;

					p_tyC0008MsgBox ACCESS ADR (tyP1040ProdSet.tyMsgBoxHide);

					//Unmask
					tyP1040ProdSet.tyProdSet.tyTableRecipe.uiMaskRtStat.0	:= TRUE;

					//Reset
					tyP1040ProdSet.tyProdSet.tyBtnSort.bRtCompl := FALSE;
				END_IF
			END_IF

		ELSE

			bUpdateP1040Table	:= TRUE;

			tyP1040ProdSet.tyProdSet.tyBtnSort.bRtCompl := FALSE;

		END_IF

	END_IF

END_ACTION
```

#### Act_OptP1040ToXML.st
```iecst
ACTION Act_OptP1040ToXML:

	IF tyP1040ProdSet.tyProdSet.tyBtnToXML.bRtCompl = TRUE THEN

		IF usiProdRcpToXMLStep = 0 THEN
			//Confirmation Message - To XML Ask
			//Mask
			fUIInRtStatOff(ADR(tyP1040ProdSet.tyProdSet.tyStringSearch.uiMaskRtStat));
			fUIInRtStatOff(ADR(tyP1040ProdSet.tyProdSet.tyTableRecipe.uiMaskRtStat));

			p_tyC0008MsgBox ACCESS ADR(tyP1040ProdSet.tyMsgBoxToXMLAsk);

			IF tyP1040ProdSet.tyMsgBoxToXMLAsk.tyBtnYes.bRtCompl = TRUE THEN
				tyP1040ProdSet.tyMsgBoxToXMLAsk.tyBtnYes.bRtCompl	:= FALSE;
				tyP1040ProdSet.tyMsgBoxToXMLAsk.tyBtnYes.bValue		:= FALSE;

				p_tyC0008MsgBox ACCESS ADR(tyP1040ProdSet.tyMsgBoxHide);

				usiProdRcpToXMLStep	:= 1;

			ELSIF tyP1040ProdSet.tyMsgBoxToXMLAsk.tyBtnNo.bRtCompl = TRUE THEN
				tyP1040ProdSet.tyMsgBoxToXMLAsk.tyBtnNo.bRtCompl	:= FALSE;
				tyP1040ProdSet.tyMsgBoxToXMLAsk.tyBtnNo.bValue		:= FALSE;

				p_tyC0008MsgBox ACCESS ADR(tyP1040ProdSet.tyMsgBoxHide);

				usiProdRcpToXMLStep	:= 99;
			END_IF

		ELSIF usiProdRcpToXMLStep = 1 THEN
			//Save Recipe To XML
			eMpProdRcpAct	:= MpProdRcpActSave;

			IF p_eMpProdRcpStat = MpProdRcpActSave AND p_eMpProdRcpStatus = Done THEN
				eMpProdRcpAct	:= MpProdRcpActIdle;

				tyP1040ProdSet.tyProdSet.tyBtnSort.bValue := FALSE;
				bRefreshProdRcpTable	:= TRUE;
				bRefreshProdRcpDetail	:= TRUE;

				usiProdRcpToXMLStep		:= 99;

			ELSIF p_eMpProdRcpStatus = Error THEN
				p_tyC0008MsgBox ACCESS ADR(tyP1040ProdSet.tyMsgBoxToXMLErr);

				IF tyP1040ProdSet.tyMsgBoxToXMLErr.tyBtnNo.bRtCompl = TRUE THEN
					tyP1040ProdSet.tyMsgBoxToXMLErr.tyBtnNo.bRtCompl	:= FALSE;
					tyP1040ProdSet.tyMsgBoxToXMLErr.tyBtnNo.bValue		:= FALSE;

					p_tyC0008MsgBox ACCESS ADR(tyP1040ProdSet.tyMsgBoxHide);

					usiProdRcpToXMLStep	:= 99;
				END_IF

			END_IF

		ELSIF usiProdRcpToXMLStep = 99 THEN
			//Complete Reset
			bRefreshProdRcpTable	:= FALSE;

			//Unmask
			fUIInRtStatHide(ADR(tyP1040ProdSet.tyProdSet.tyStringSearch.uiMaskRtStat));
			fUIInRtStatHide(ADR(tyP1040ProdSet.tyProdSet.tyTableRecipe.uiMaskRtStat));

			tyP1040ProdSet.tyProdSet.tyBtnToXML.bRtCompl	:= FALSE;
			tyP1040ProdSet.tyProdSet.tyBtnToXML.bValue		:= FALSE;

			usiProdRcpToXMLStep	:= 0;

		END_IF

	END_IF

END_ACTION
```

#### Act_OptP1040FromXML.st
```iecst
ACTION Act_OptP1040FromXML:

	IF tyP1040ProdSet.tyProdSet.tyBtnFromXML.bRtCompl = TRUE THEN

		IF usiProdRcpFromXMLStep = 0 THEN
			//Confirmation Message - From XML Ask
			//Mask
			fUIInRtStatOff(ADR(tyP1040ProdSet.tyProdSet.tyStringSearch.uiMaskRtStat));
			fUIInRtStatOff(ADR(tyP1040ProdSet.tyProdSet.tyTableRecipe.uiMaskRtStat));

			p_tyC0008MsgBox ACCESS ADR(tyP1040ProdSet.tyMsgBoxFromXMLAsk);

			IF tyP1040ProdSet.tyMsgBoxFromXMLAsk.tyBtnYes.bRtCompl = TRUE THEN
				tyP1040ProdSet.tyMsgBoxFromXMLAsk.tyBtnYes.bRtCompl	:= FALSE;
				tyP1040ProdSet.tyMsgBoxFromXMLAsk.tyBtnYes.bValue	:= FALSE;

				p_tyC0008MsgBox ACCESS ADR(tyP1040ProdSet.tyMsgBoxHide);

				usiProdRcpFromXMLStep	:= 1;

			ELSIF tyP1040ProdSet.tyMsgBoxFromXMLAsk.tyBtnNo.bRtCompl = TRUE THEN
				tyP1040ProdSet.tyMsgBoxFromXMLAsk.tyBtnNo.bRtCompl	:= FALSE;
				tyP1040ProdSet.tyMsgBoxFromXMLAsk.tyBtnNo.bValue	:= FALSE;

				p_tyC0008MsgBox ACCESS ADR(tyP1040ProdSet.tyMsgBoxHide);

				usiProdRcpFromXMLStep	:= 99;
			END_IF

		ELSIF usiProdRcpFromXMLStep = 1 THEN
			//Load Recipe From XML
			eMpProdRcpAct	:= MpProdRcpActLoad;

			IF p_eMpProdRcpStat = MpProdRcpActLoad AND p_eMpProdRcpStatus = Done THEN
				eMpProdRcpAct	:= MpProdRcpActIdle;

				tyP1040ProdSet.tyProdSet.tyBtnSort.bValue      := FALSE;
				tyP1040ProdSet.tyProdSet.tyStringSearch.sValue := '';
				bRefreshProdRcpTable	:= TRUE;
				bRefreshProdRcpDetail	:= TRUE;

				usiProdRcpFromXMLStep	:= 2;

			ELSIF p_eMpProdRcpStatus = Error THEN
				p_tyC0008MsgBox ACCESS ADR(tyP1040ProdSet.tyMsgBoxFromXMLErr);

				IF tyP1040ProdSet.tyMsgBoxFromXMLErr.tyBtnNo.bRtCompl = TRUE THEN
					tyP1040ProdSet.tyMsgBoxFromXMLErr.tyBtnNo.bRtCompl	:= FALSE;
					tyP1040ProdSet.tyMsgBoxFromXMLErr.tyBtnNo.bValue	:= FALSE;

					p_tyC0008MsgBox ACCESS ADR(tyP1040ProdSet.tyMsgBoxHide);

					usiProdRcpFromXMLStep	:= 99;
				END_IF

			END_IF

		ELSIF usiProdRcpFromXMLStep = 2 THEN
			//Save Product Recipe List
			eProdRcpAct	:= ProdRcpActSaveList;

			IF p_eProdRcpStat = ProdRcpActSaveList AND p_eProdRcpStatus = Done THEN
				eProdRcpAct	:= ProdRcpActIdle;

				usiProdRcpFromXMLStep	:= 99;

			ELSIF p_eProdRcpStatus = Error THEN
				p_tyC0008MsgBox ACCESS ADR(tyP1040ProdSet.tyMsgBoxSaveListErr);

				IF tyP1040ProdSet.tyMsgBoxSaveListErr.tyBtnNo.bRtCompl = TRUE THEN
					tyP1040ProdSet.tyMsgBoxSaveListErr.tyBtnNo.bRtCompl	:= FALSE;
					tyP1040ProdSet.tyMsgBoxSaveListErr.tyBtnNo.bValue	:= FALSE;

					p_tyC0008MsgBox ACCESS ADR(tyP1040ProdSet.tyMsgBoxHide);

					usiProdRcpFromXMLStep	:= 99;
				END_IF

			END_IF

		ELSIF usiProdRcpFromXMLStep = 99 THEN
			//Complete Reset
			bRefreshProdRcpTable	:= FALSE;

			//Unmask
			fUIInRtStatHide(ADR(tyP1040ProdSet.tyProdSet.tyStringSearch.uiMaskRtStat));
			fUIInRtStatHide(ADR(tyP1040ProdSet.tyProdSet.tyTableRecipe.uiMaskRtStat));

			tyP1040ProdSet.tyProdSet.tyBtnFromXML.bRtCompl	:= FALSE;
			tyP1040ProdSet.tyProdSet.tyBtnFromXML.bValue	:= FALSE;

			usiProdRcpFromXMLStep	:= 0;

		END_IF

	END_IF

END_ACTION
```

#### Act_EntP1050Disp.st
```iecst
ACTION Act_EntP1050Disp:

	//Access Address
	p_tyC0005Main ACCESS ADR(tyCommon.tyMain);

	p_tyC0006Set ACCESS ADR(tyCommon.tySet);

	p_tyC0007Notif ACCESS ADR(tyCommon.tyNotif);

	p_tyC0008MsgBox ACCESS ADR(tyP1050LFSet.tyMsgBoxHide);

	p_tyC0009Info ACCESS ADR(tyCommon.tyInfo);

	p_tyP1050LFSetLdrEdit ACCESS ADR(tyP1050LFSet.tyLdrEdit);
	p_tyP1050LFSetLdr ACCESS ADR(tyP1050LFSet.tyLdr);

END_ACTION
```

#### Act_OptP1050Edit.st
```iecst
ACTION Act_OptP1050Edit:

	IF tyP1050LFSet.tyLdr.tyBtnEdit.bRtCompl = TRUE THEN

		FOR i := 1 TO UDINT_TO_UINT(c_diLFClntNum) DO
			IF tyMcParamWr.a_sLFIPAddr[i] = '' THEN
				uiLFStartEditNo	:= i;
				EXIT;
			END_IF
		END_FOR

		tyP1050LFSet.tyLdr.tyBtnEdit.bRtCompl	:= FALSE;
		tyP1050LFSet.tyLdr.tyBtnEdit.bValue		:= TRUE;

		fUIInRtStatOff(ADR(tyP1050LFSet.tyLdrEdit.tyLyr.uiRtStat));
		fUIInRtStatHide(ADR(tyP1050LFSet.tyLdr.tyLyr.uiRtStat));

		tyP1050LFSet.tyLdrEdit.tyNumMcNum.diValue		:= STRING_TO_DINT(tyP1050LFSet.tyLdr.tyTable1List.a_tyStringDataCol0[tyP1050Table.uiSelectedRow].sValue);
		tyP1050LFSet.tyLdrEdit.tyStringIPAddr.sValue	:= tyP1050LFSet.tyLdr.tyTable1List.a_tyStringDataCol2[tyP1050Table.uiSelectedRow].sValue;

	ELSIF tyP1050LFSet.tyLdr.tyBtnEdit.bValue = TRUE THEN

		IF tyP1050LFSet.tyLdrEdit.tyBtnOk.bRtCompl = TRUE THEN

			IF fIPValid(tyP1050LFSet.tyLdrEdit.tyStringIPAddr.sValue , ADR(a_iIPPart1)) = TRUE AND bCheckDone = FALSE THEN
				FOR i := 1 TO UDINT_TO_UINT(c_diLFClntNum) DO
					IF i <>  tyP1050Table.uiTablePos + tyP1050Table.uiSelectedRow - 1 THEN
						fIPValid(p_tyMcParamCurr.a_sLFIPAddr[i] , ADR(a_iIPPart2));

						IF (a_iIPPart1[1] = a_iIPPart2[1] AND a_iIPPart1[2] = a_iIPPart2[2] AND a_iIPPart1[3] = a_iIPPart2[3] AND a_iIPPart1[4] = a_iIPPart2[4])
							AND (tyP1050LFSet.tyLdrEdit.tyStringIPAddr.sValue <> '') THEN

							bIPDuplicate	:= TRUE;
							EXIT;

						END_IF
					END_IF
				END_FOR
				bCheckDone := TRUE;
			END_IF

			IF fIPValid(tyP1050LFSet.tyLdrEdit.tyStringIPAddr.sValue , ADR(a_iIPPart1)) = FALSE THEN
				p_tyC0008MsgBox ACCESS ADR(tyP1050LFSet.tyMsgBoxIPAddrInvalid);

				IF tyP1050LFSet.tyMsgBoxIPAddrInvalid.tyBtnNo.bRtCompl = TRUE THEN
					tyP1050LFSet.tyMsgBoxIPAddrInvalid.tyBtnNo.bRtCompl	:= FALSE;
					tyP1050LFSet.tyMsgBoxIPAddrInvalid.tyBtnNo.bValue	:= FALSE;

					p_tyC0008MsgBox ACCESS ADR(tyP1050LFSet.tyMsgBoxHide);

					tyP1050LFSet.tyLdrEdit.tyBtnOk.bRtCompl	:= FALSE;
					tyP1050LFSet.tyLdrEdit.tyBtnOk.bValue	:= FALSE;
					bCheckDone := FALSE;
				END_IF

			ELSIF bIPDuplicate = TRUE THEN
				p_tyC0008MsgBox ACCESS ADR(tyP1050LFSet.tyMsgBoxIPAddrDuplicate);

				IF tyP1050LFSet.tyMsgBoxIPAddrDuplicate.tyBtnNo.bRtCompl = TRUE THEN
					tyP1050LFSet.tyMsgBoxIPAddrDuplicate.tyBtnNo.bRtCompl	:= FALSE;
					tyP1050LFSet.tyMsgBoxIPAddrDuplicate.tyBtnNo.bValue		:= FALSE;

					p_tyC0008MsgBox ACCESS ADR(tyP1050LFSet.tyMsgBoxHide);

					bIPDuplicate							:= FALSE;
					tyP1050LFSet.tyLdrEdit.tyBtnOk.bRtCompl	:= FALSE;
					tyP1050LFSet.tyLdrEdit.tyBtnOk.bValue	:= FALSE;
					bCheckDone := FALSE;
				END_IF
			ELSE
				IF tyP1050LFSet.tyLdr.tyTable1List.a_tyStringDataCol2[tyP1050Table.uiSelectedRow].sValue = '' THEN
					tyMcParamWr.a_sLFIPAddr[uiLFStartEditNo]	:= tyP1050LFSet.tyLdrEdit.tyStringIPAddr.sValue;

					eMcParamAct	:= McParamActWrite;

					IF p_eMcParamStat = McParamActWrite AND p_eMcParamStatus = Done THEN
						eMcParamAct	:= McParamActIdle;

						tyP1050LFSet.tyLdr.tyTable1List.a_tyStringDataCol2[uiLFStartEditNo].sValue		:= tyP1050LFSet.tyLdrEdit.tyStringIPAddr.sValue;

						IF tyP1050LFSet.tyLdrEdit.tyStringIPAddr.sValue = '0000' THEN
							tyP1050LFSet.tyLdr.tyTable1List.a_tyTxtDataCol3[uiLFStartEditNo].usiValueIdx	:= 3;
						ELSE
							tyP1050LFSet.tyLdr.tyTable1List.a_tyTxtDataCol3[uiLFStartEditNo].usiValueIdx	:= 1;
						END_IF

						//LF Control
						FOR i := 1 TO c_uiP1050TableSize DO
							tyP0700LFCtrl.tyLdr.tyTable1List.a_tyStringDataCol0[i].sValue	:= UINT_TO_STRING(tyP0700Table.uiTablePos + i - 1);
							tyP0700LFCtrl.tyLdr.tyTable1List.a_tyStringDataCol2[i].sValue	:= p_tyMcParamCurr.a_sLFIPAddr[tyP0700Table.uiTablePos + i - 1];
						END_FOR

						tyP1050LFSet.tyLdrEdit.tyBtnOk.bRtCompl	:= FALSE;
						tyP1050LFSet.tyLdrEdit.tyBtnOk.bValue	:= FALSE;
						tyP1050LFSet.tyLdr.tyBtnEdit.bValue		:= FALSE;
						bCheckDone								:= FALSE;

						bUpdateP1050Table	:=TRUE;

						fUIInRtStatHide(ADR(tyP1050LFSet.tyLdrEdit.tyLyr.uiRtStat));
						fUIInRtStatOff(ADR(tyP1050LFSet.tyLdr.tyLyr.uiRtStat));

					ELSIF p_eMcParamStatus = Error THEN
						p_tyC0008MsgBox ACCESS ADR(tyP1050LFSet.tyMsgBoxSaveErr);

						IF tyP1050LFSet.tyMsgBoxSaveErr.tyBtnNo.bRtCompl = TRUE THEN
							tyP1050LFSet.tyMsgBoxSaveErr.tyBtnNo.bRtCompl	:= FALSE;
							tyP1050LFSet.tyMsgBoxSaveErr.tyBtnNo.bValue		:= FALSE;

							p_tyC0008MsgBox ACCESS ADR(tyP1050LFSet.tyMsgBoxHide);

							//Recover
							tyMcParamWr	:= p_tyMcParamCurr;

							tyP1050LFSet.tyLdrEdit.tyBtnOk.bRtCompl	:= FALSE;
							tyP1050LFSet.tyLdrEdit.tyBtnOk.bValue	:= FALSE;
							tyP1050LFSet.tyLdr.tyBtnEdit.bValue		:= FALSE;
							bCheckDone								:=FALSE;

							fUIInRtStatHide(ADR(tyP1050LFSet.tyLdrEdit.tyLyr.uiRtStat));
							fUIInRtStatOff(ADR(tyP1050LFSet.tyLdr.tyLyr.uiRtStat));
						END_IF
					END_IF
				ELSE
					tyMcParamWr.a_sLFIPAddr[tyP1050Table.uiTablePos + tyP1050Table.uiSelectedRow - 1]	:= tyP1050LFSet.tyLdrEdit.tyStringIPAddr.sValue;

					eMcParamAct	:= McParamActWrite;

					IF p_eMcParamStat = McParamActWrite AND p_eMcParamStatus = Done THEN
						eMcParamAct	:= McParamActIdle;

						tyP1050LFSet.tyLdr.tyTable1List.a_tyStringDataCol2[tyP1050Table.uiSelectedRow].sValue		:= tyP1050LFSet.tyLdrEdit.tyStringIPAddr.sValue;

						IF tyP1050LFSet.tyLdrEdit.tyStringIPAddr.sValue = '0000' THEN
							tyP1050LFSet.tyLdr.tyTable1List.a_tyTxtDataCol3[tyP1050Table.uiSelectedRow].usiValueIdx	:= 3;
						ELSE
							tyP1050LFSet.tyLdr.tyTable1List.a_tyTxtDataCol3[ tyP1050Table.uiSelectedRow].usiValueIdx	:= 1;
						END_IF

						//LF Control
						FOR i := 1 TO c_uiP1050TableSize DO
							tyP0700LFCtrl.tyLdr.tyTable1List.a_tyStringDataCol0[i].sValue	:= UINT_TO_STRING(tyP0700Table.uiTablePos + i - 1);
							tyP0700LFCtrl.tyLdr.tyTable1List.a_tyStringDataCol2[i].sValue	:= p_tyMcParamCurr.a_sLFIPAddr[tyP0700Table.uiTablePos + i - 1];
						END_FOR

						tyP1050LFSet.tyLdrEdit.tyBtnOk.bRtCompl	:= FALSE;
						tyP1050LFSet.tyLdrEdit.tyBtnOk.bValue	:= FALSE;
						tyP1050LFSet.tyLdr.tyBtnEdit.bValue		:= FALSE;
						bCheckDone								:= FALSE;

						fUIInRtStatHide(ADR(tyP1050LFSet.tyLdrEdit.tyLyr.uiRtStat));
						fUIInRtStatOff(ADR(tyP1050LFSet.tyLdr.tyLyr.uiRtStat));

					ELSIF p_eMcParamStatus = Error THEN

						p_tyC0008MsgBox ACCESS ADR(tyP1050LFSet.tyMsgBoxSaveErr);

						IF tyP1050LFSet.tyMsgBoxSaveErr.tyBtnNo.bRtCompl = TRUE THEN
							tyP1050LFSet.tyMsgBoxSaveErr.tyBtnNo.bRtCompl	:= FALSE;
							tyP1050LFSet.tyMsgBoxSaveErr.tyBtnNo.bValue		:= FALSE;

							p_tyC0008MsgBox ACCESS ADR(tyP1050LFSet.tyMsgBoxHide);

							//Recover
							tyMcParamWr	:= p_tyMcParamCurr;

							tyP1050LFSet.tyLdrEdit.tyBtnOk.bRtCompl	:= FALSE;
							tyP1050LFSet.tyLdrEdit.tyBtnOk.bValue	:= FALSE;
							tyP1050LFSet.tyLdr.tyBtnEdit.bValue		:= FALSE;
							bCheckDone								:=FALSE;

							fUIInRtStatHide(ADR(tyP1050LFSet.tyLdrEdit.tyLyr.uiRtStat));
							fUIInRtStatOff(ADR(tyP1050LFSet.tyLdr.tyLyr.uiRtStat));
						END_IF
					END_IF
				END_IF
			END_IF

		ELSIF tyP1050LFSet.tyLdrEdit.tyBtnCancel.bRtCompl = TRUE THEN
			tyP1050LFSet.tyLdrEdit.tyBtnCancel.bRtCompl	:= FALSE;
			tyP1050LFSet.tyLdrEdit.tyBtnCancel.bValue	:= FALSE;
			tyP1050LFSet.tyLdr.tyBtnEdit.bValue			:= FALSE;

			fUIInRtStatHide(ADR(tyP1050LFSet.tyLdrEdit.tyLyr.uiRtStat));
			fUIInRtStatOff(ADR(tyP1050LFSet.tyLdr.tyLyr.uiRtStat));
		END_IF
	END_IF

	IF bLFSettingAutoFill THEN

		iIPExtract:= LEN(p_sHWInfoIPAddr)-10;
		sLFSettingCurrentIP := RIGHT(p_sHWInfoIPAddr,iIPExtract);
		iLFSettingCurrentIP	:= STRING_TO_INT(sLFSettingCurrentIP);

		FOR i:= 1 TO 20 DO
			sLFSettingAutoFill	:='192.168.0.';
			sLFSettingTemp		:=UINT_TO_STRING(iLFSettingCurrentIP+(i*2)-2);
			sLFSettingAutoFill	:=CONCAT(sLFSettingAutoFill,sLFSettingTemp);
			tyMcParamWr.a_sLFIPAddr[i]:= sLFSettingAutoFill;
			tyMcParamWr.a_bLFOnline[i]:= FALSE;
		END_FOR

		eMcParamAct	:= McParamActWrite;

		IF p_eMcParamStat = McParamActWrite AND p_eMcParamStatus = Done THEN
			eMcParamAct	:= McParamActIdle;
			bUpdateP1050Table	:= TRUE;
			bLFSettingAutoFill	:= FALSE;
		ELSIF p_eMcParamStatus = Error THEN
			//Recover
			tyMcParamWr	:= p_tyMcParamCurr;
			bUpdateP1050Table	:= TRUE;
			bLFSettingAutoFill	:= FALSE;
		END_IF

	END_IF

	IF bLFSettingAutoClear THEN
		FOR i:= 1 TO 20 DO
			tyMcParamWr.a_sLFIPAddr[i]:= '';
			tyMcParamWr.a_bLFOnline[i]:= FALSE;
		END_FOR

		eMcParamAct	:= McParamActWrite;

		IF p_eMcParamStat = McParamActWrite AND p_eMcParamStatus = Done THEN
			eMcParamAct	:= McParamActIdle;
			bUpdateP1050Table	:= TRUE;
			bLFSettingAutoClear	:= FALSE;
		ELSIF p_eMcParamStatus = Error THEN
			//Recover
			tyMcParamWr	:= p_tyMcParamCurr;
			bUpdateP1050Table	:= TRUE;
			bLFSettingAutoClear	:= FALSE;
		END_IF

	END_IF

END_ACTION
```

#### Act_OptP1050Delete.st
```iecst
ACTION Act_OptP1050Delete:

	IF tyP1050LFSet.tyLdr.tyBtnDelete.bRtCompl = TRUE THEN
		IF usiDelMcDetailsStep = 0 THEN
			p_tyC0008MsgBox ACCESS ADR(tyP1050LFSet.tyMsgBoxDelAsk);

			IF tyP1050LFSet.tyMsgBoxDelAsk.tyBtnYes.bRtCompl = TRUE THEN
				tyP1050LFSet.tyMsgBoxDelAsk.tyBtnYes.bRtCompl	:= FALSE;
				tyP1050LFSet.tyMsgBoxDelAsk.tyBtnYes.bValue		:= FALSE;

				p_tyC0008MsgBox ACCESS ADR(tyP1050LFSet.tyMsgBoxHide);

				usiDelMcDetailsStep	:= 1;

			ELSIF tyP1050LFSet.tyMsgBoxDelAsk.tyBtnNo.bRtCompl = TRUE THEN
				tyP1050LFSet.tyMsgBoxDelAsk.tyBtnNo.bRtCompl	:= FALSE;
				tyP1050LFSet.tyMsgBoxDelAsk.tyBtnNo.bValue		:= FALSE;

				p_tyC0008MsgBox ACCESS ADR(tyP1050LFSet.tyMsgBoxHide);

				tyP1050LFSet.tyLdr.tyBtnDelete.bRtCompl			:= FALSE;
				tyP1050LFSet.tyLdr.tyBtnDelete.bValue			:= FALSE;
			END_IF

		ELSIF usiDelMcDetailsStep = 1 THEN
			tyMcParamWr.a_sLFIPAddr[tyP1050Table.uiTablePos + tyP1050Table.uiSelectedRow - 1]	:= '';
			tyMcParamWr.a_bLFOnline[tyP1050Table.uiTablePos + tyP1050Table.uiSelectedRow - 1]	:= FALSE;

			eMcParamAct	:= McParamActWrite;

			IF p_eMcParamStat = McParamActWrite AND p_eMcParamStatus = Done THEN
				eMcParamAct	:= McParamActIdle;

				tyP1050LFSet.tyLdr.tyTable1List.a_tyStringDataCol2[tyP1050Table.uiSelectedRow].sValue	:= '';
				tyP1050LFSet.tyLdr.tyTable1List.a_tyTxtDataCol3[tyP1050Table.uiSelectedRow].usiValueIdx	:= 0;

				//UIP0700 LF Control
				FOR i := 1 TO c_uiP1050TableSize DO
					tyP0700LFCtrl.tyLdr.tyTable1List.a_tyStringDataCol0[i].sValue	:= UINT_TO_STRING(tyP0700Table.uiTablePos + i - 1);
					tyP0700LFCtrl.tyLdr.tyTable1List.a_tyStringDataCol2[i].sValue	:= p_tyMcParamCurr.a_sLFIPAddr[tyP0700Table.uiTablePos + i - 1];
				END_FOR

				usiDelMcDetailsStep		:= 0;

				tyP1050LFSet.tyLdr.tyBtnDelete.bRtCompl				:= FALSE;
				tyP1050LFSet.tyLdr.tyBtnDelete.bValue				:= FALSE;

			ELSIF p_eMcParamStatus = Error THEN
				p_tyC0008MsgBox ACCESS ADR(tyP1050LFSet.tyMsgBoxSaveErr);

				IF tyP1050LFSet.tyMsgBoxSaveErr.tyBtnNo.bRtCompl = TRUE THEN
					tyP1050LFSet.tyMsgBoxSaveErr.tyBtnNo.bRtCompl	:= FALSE;
					tyP1050LFSet.tyMsgBoxSaveErr.tyBtnNo.bValue		:= FALSE;

					p_tyC0008MsgBox ACCESS ADR(tyP1050LFSet.tyMsgBoxHide);

					//Recover
					tyMcParamWr	:= p_tyMcParamCurr;

					usiDelMcDetailsStep	:= 0;

					tyP1050LFSet.tyLdr.tyBtnDelete.bRtCompl			:= FALSE;
					tyP1050LFSet.tyLdr.tyBtnDelete.bValue			:= FALSE;
				END_IF
			END_IF
		END_IF
	END_IF

END_ACTION
```

#### Act_OptP1050Table.st
```iecst
ACTION Act_OptP1050Table:

	//Call Table FB
	fbP1050Table.sVisuNm			:= tyP1050Table.sVisuNm;
	fbP1050Table.udiWorkAreaStartX	:= 96;
	fbP1050Table.udiWorkAreaEndX	:= 554;
	fbP1050Table.udiWorkAreaStartY	:= 75;
	fbP1050Table.udiWorkAreaEndY	:= 455;
	fbP1050Table.udiMinXDist		:= 20;
	fbP1050Table.udiMinYDist		:= 20;
	fbP1050Table.uiSlideScale		:= c_uiP1050TableSize;
	fbP1050Table.iTotalData			:= UDINT_TO_INT(c_diLFClntNum);
	fbP1050Table.iTotalRow			:= c_uiP1050TableSize;
	fbP1050Table(uiSliderStatus := tyP1050LFSet.tyLdr.tyTable1List.tyUISlider.uiRtStat , a_tyUIHotspot := tyP1050LFSet.tyLdr.tyTable1List.a_tyHotspot , uiTablePos := tyP1050Table.uiTablePos , iSliderPos := tyP1050LFSet.tyLdr.tyTable1List.tyUISlider.iValue);

	tyP1050Table.uiSelectedRow		:= fbP1050Table.uiSelectedRow;
	tyP1050Table.bTableActive		:= fbP1050Table.bTableActive;
	tyP1050Table.bSliderActive		:= fbP1050Table.bSliderActive;

	//Table Content
	IF tyP1050Table.bTableActive = TRUE OR tyP1050Table.bSliderActive = TRUE OR usiTableShftStep = 3 THEN
		FOR i := 1 TO c_uiP1050TableSize DO
			tyP1050LFSet.tyLdr.tyTable1List.a_tyStringDataCol0[i].sValue			:= UINT_TO_STRING(tyP1050Table.uiTablePos + i - 1);
			tyP1050LFSet.tyLdr.tyTable1List.a_tyStringDataCol2[i].sValue			:= p_tyMcParamCurr.a_sLFIPAddr[tyP1050Table.uiTablePos + i - 1];

			IF tyP1050LFSet.tyLdr.tyTable1List.a_tyStringDataCol2[i].sValue = '' THEN
				tyP1050LFSet.tyLdr.tyTable1List.a_tyTxtDataCol3[i].usiValueIdx	:= 0;
			ELSIF tyP1050LFSet.tyLdr.tyTable1List.a_tyStringDataCol2[i].sValue = '0000' THEN
				tyP1050LFSet.tyLdr.tyTable1List.a_tyTxtDataCol3[i].usiValueIdx	:= 3;
			ELSE
				tyP1050LFSet.tyLdr.tyTable1List.a_tyTxtDataCol3[i].usiValueIdx	:= (BOOL_TO_USINT(p_tyMcParamCurr.a_bLFOnline[tyP1050Table.uiTablePos + i - 1])) + 1;
			END_IF

		END_FOR

	END_IF

	//Selected Row
	IF tyP1050Table.uiSelectedRow <> tyP1050Table.uiSelectedRowOld THEN
		FOR i := 1 TO c_uiP1050TableSize DO
			IF tyP1050Table.uiSelectedRow = i THEN
				tyP1050LFSet.tyLdr.tyTable1List.a_tyStringDataCol2[i].usiColor	:= 1;
				tyP1050LFSet.tyLdr.tyTable1List.a_tyTxtDataCol3[i].usiColor		:= 1;

			ELSE
				tyP1050LFSet.tyLdr.tyTable1List.a_tyStringDataCol2[i].usiColor	:= 0;
				tyP1050LFSet.tyLdr.tyTable1List.a_tyTxtDataCol3[i].usiColor		:= 0;

			END_IF

		END_FOR

		tyP1050Table.uiSelectedRowOld	:= tyP1050Table.uiSelectedRow;

	END_IF

END_ACTION
```

#### Act_OptP1050Keypad.st
```iecst
ACTION Act_OptP1050Keypad:

	IF fUIOutRtStatTPIsOpen(ADR(tyP1050LFSet.tyLdrEdit.tyStringIPAddr.uiRtStat)) THEN
		tyProperty.tyKeypad.tyStringTitle.sKeypadTitle	:= tyP1050LFSet.tyLdrEdit.tyStringIPAddr.sKeypadTitle;

	ELSIF fUIOutRtStatTPIsOpen(ADR(tyP1050LFSet.tyLdr.tyNumAfterOven.uiRtStat)) THEN
		tyProperty.tyKeypad.tyStringTitle.sKeypadTitle	:= tyP1050LFSet.tyLdr.tyNumAfterOven.sKeypadTitle;

	ELSIF fUIOutRtStatTPIsOpen(ADR(tyP1050LFSet.tyLdr.tyNumBeforeOven.uiRtStat)) THEN
		tyProperty.tyKeypad.tyStringTitle.sKeypadTitle	:= tyP1050LFSet.tyLdr.tyNumBeforeOven.sKeypadTitle;

	ELSE
		tyProperty.tyKeypad.tyStringTitle.sKeypadTitle	:= '';

	END_IF

END_ACTION
```

#### Act_OptP1050Oven.st
```iecst
ACTION Act_OptP1050Oven:

	IF tyP1050LFSet.tyLdr.tyNumBeforeOven.bRtCompl = TRUE OR tyP1050LFSet.tyLdr.tyNumAfterOven.bRtCompl = TRUE THEN

		tyMcParamWr.diLFMcIdxBeforeOven	:= tyP1050LFSet.tyLdr.tyNumBeforeOven.diValue;
		tyMcParamWr.diLFMcIdxAfterOven	:= tyP1050LFSet.tyLdr.tyNumAfterOven.diValue;

		eMcParamAct		:= McParamActWrite;

		IF p_eMcParamStat = McParamActWrite AND p_eMcParamStatus = Done THEN
			eMcParamAct		:= McParamActIdle;

			//BackUp Param
			tyP1050LFSet.tyLdrBkUp	:= tyP1050LFSet.tyLdr;

			tyP1050LFSet.tyLdr.tyNumBeforeOven.bRtCompl := FALSE;
			tyP1050LFSet.tyLdr.tyNumAfterOven.bRtCompl  := FALSE;

		ELSIF p_eMcParamStatus = Error THEN
			p_tyC0008MsgBox ACCESS ADR(tyP1050LFSet.tyMsgBoxSaveErr);

			IF tyP1050LFSet.tyMsgBoxSaveErr.tyBtnNo.bRtCompl = TRUE THEN
				tyP1050LFSet.tyMsgBoxSaveErr.tyBtnNo.bRtCompl 	:= FALSE;
				tyP1050LFSet.tyMsgBoxSaveErr.tyBtnNo.bValue		:= FALSE;

				tyP1050LFSet.tyLdr.tyNumBeforeOven.bRtCompl := FALSE;
				tyP1050LFSet.tyLdr.tyNumAfterOven.bRtCompl  := FALSE;

				p_tyC0008MsgBox ACCESS ADR(tyP1050LFSet.tyMsgBoxHide);

				// Restore Param
				tyP1050LFSet.tyLdr		:= tyP1050LFSet.tyLdrBkUp;
				tyMcParamWr				:= p_tyMcParamCurr;

			END_IF

		END_IF

	END_IF

END_ACTION
```

#### Act_EntP1080Disp.st
```iecst
ACTION Act_EntP1080Disp:

	//Access Address
	p_tyC0005Main ACCESS ADR(tyCommon.tyMain);

	p_tyC0007Notif ACCESS ADR(tyCommon.tyNotif);

	p_tyC0008MsgBox ACCESS ADR(tyP1080UsrMgmt.tyMsgBoxHide);

	p_tyC0009Info ACCESS ADR(tyCommon.tyInfo);

	p_tyP1080UsrMgmt ACCESS ADR(tyP1080UsrMgmt.tyUsrMgmt);
	p_tyP1080UsrMgmtAct ACCESS ADR(tyP1080UsrMgmt.tyCreate);

	//Display
	fUIInRtStatHide(ADR(tyP1080UsrMgmt.tyCreate.tyLyr.uiRtStat));
	fUIInRtStatOff(ADR(tyP1080UsrMgmt.tyUsrMgmt.tyLyr.uiRtStat));

	IF tyP1080UsrMgmt.tyUsrMgmt.tyDrpDnLvl.usiValueIdx > tyP1080UsrMgmt.tyUsrMgmt.tyDrpDnLvl.usiValueMaxIdx THEN
		tyP1080UsrMgmt.tyUsrMgmt.tyDrpDnLvl.usiValueIdx	:= 0;
		tyP1080UsrMgmt.tyUsrMgmt.tyDrpDnLvl.bRtCompl	:= TRUE;
	END_IF

END_ACTION
```

#### Act_OptP1080Keypad.st
```iecst
ACTION Act_OptP1080Keypad:

	IF fUIOutRtStatTPIsOpen(ADR(tyP1080UsrMgmt.tyCreate.tyStringUsrNm.uiRtStat)) = TRUE THEN
		tyProperty.tyKeypad.tyStringTitle.sKeypadTitle	:= tyP1080UsrMgmt.tyCreate.tyStringUsrNm.sKeypadTitle;

	ELSIF fUIOutRtStatTPIsOpen(ADR(tyP1080UsrMgmt.tyCreate.tyStringPw.uiRtStat)) = TRUE THEN
		tyProperty.tyKeypad.tyStringTitle.sKeypadTitle	:= tyP1080UsrMgmt.tyCreate.tyStringPw.sKeypadTitle;

	ELSIF fUIOutRtStatTPIsOpen(ADR(tyP1080UsrMgmt.tyEdit.tyStringPw.uiRtStat)) = TRUE THEN
		tyProperty.tyKeypad.tyStringTitle.sKeypadTitle	:= tyP1080UsrMgmt.tyCreate.tyStringPw.sKeypadTitle;

	ELSE
		tyProperty.tyKeypad.tyStringTitle.sKeypadTitle	:= '';

	END_IF

END_ACTION
```

#### Act_OptP1080Table.st
```iecst
ACTION Act_OptP1080Table:

	fbP1080Table.sVisuNm			:= tyP1080Table.sVisuNm;
	fbP1080Table.udiWorkAreaStartX	:= 50;
	fbP1080Table.udiWorkAreaEndX	:= 497;
	fbP1080Table.udiWorkAreaStartY	:= 109;
	fbP1080Table.udiWorkAreaEndY	:= 458;
	fbP1080Table.udiMinXDist		:= 20;
	fbP1080Table.udiMinYDist		:= 20;
	fbP1080Table.uiSlideScale		:= c_uiP1080TableSize;
	fbP1080Table.iTotalData			:= UDINT_TO_INT(c_udiUsrMgmtMax);
	fbP1080Table.iTotalRow			:= c_uiP1080TableSize;
	fbP1080Table(uiSliderStatus := tyP1080UsrMgmt.tyUsrMgmt.tyTableList.tyUISlider.uiRtStat , a_tyUIHotspot := tyP1080UsrMgmt.tyUsrMgmt.tyTableList.a_tyHotspot , uiTablePos := tyP1080Table.uiTablePos , iSliderPos := tyP1080UsrMgmt.tyUsrMgmt.tyTableList.tyUISlider.iValue);

	tyP1080Table.uiSelectedRow		:= fbP1080Table.uiSelectedRow;
	tyP1080Table.bTableActive		:= fbP1080Table.bTableActive;
	tyP1080Table.bSliderActive		:= fbP1080Table.bSliderActive;

	//Table Content
	IF tyP1080Table.bTableActive = TRUE OR tyP1080Table.bSliderActive = TRUE OR bRefreshUsrMgmtTable = TRUE THEN
		FOR i := 1 TO c_uiP1080TableSize DO

			tyP1080UsrMgmt.tyUsrMgmt.tyTableList.a_tyStringDataCol0[i].sValue				:= UINT_TO_STRING(tyP1080Table.uiTablePos + i - 1);

			CASE tyP1080UsrMgmt.tyUsrMgmt.tyDrpDnLvl.usiValueIdx OF
				//User All
				0:
					tyP1080UsrMgmt.tyUsrMgmt.tyTableList.a_tyStringDataCol1[i].sValue		:= p_tyUsrMgmtAllList[tyP1080Table.uiTablePos + i - 1].sUsrNm;
					tyP1080UsrMgmt.tyUsrMgmt.tyTableList.a_tyTxtDataCol3[i].usiValueIdx		:= DINT_TO_USINT(p_tyUsrMgmtAllList[tyP1080Table.uiTablePos + i - 1].eUsrLvl + 1);
				//User Level 2
				1:
					tyP1080UsrMgmt.tyUsrMgmt.tyTableList.a_tyStringDataCol1[i].sValue		:= p_tyUsrMgmtLv2List[tyP1080Table.uiTablePos + i - 1].sUsrNm;
					tyP1080UsrMgmt.tyUsrMgmt.tyTableList.a_tyTxtDataCol3[i].usiValueIdx		:= DINT_TO_USINT(p_tyUsrMgmtLv2List[tyP1080Table.uiTablePos + i - 1].eUsrLvl + 1);
				//User Level 3
				2:
					tyP1080UsrMgmt.tyUsrMgmt.tyTableList.a_tyStringDataCol1[i].sValue		:= p_tyUsrMgmtLv3List[tyP1080Table.uiTablePos + i - 1].sUsrNm;
					tyP1080UsrMgmt.tyUsrMgmt.tyTableList.a_tyTxtDataCol3[i].usiValueIdx		:= DINT_TO_USINT(p_tyUsrMgmtLv3List[tyP1080Table.uiTablePos + i - 1].eUsrLvl + 1);
				//User Admin
				3:
					tyP1080UsrMgmt.tyUsrMgmt.tyTableList.a_tyStringDataCol1[i].sValue		:= p_tyUsrMgmtAdminList[tyP1080Table.uiTablePos + i - 1].sUsrNm;
					tyP1080UsrMgmt.tyUsrMgmt.tyTableList.a_tyTxtDataCol3[i].usiValueIdx		:= DINT_TO_USINT(p_tyUsrMgmtAdminList[tyP1080Table.uiTablePos + i - 1].eUsrLvl + 1);
			END_CASE
		END_FOR
		bRefreshUsrMgmtTable 			:= FALSE;
	END_IF

	IF tyP1080UsrMgmt.tyUsrMgmt.tyDrpDnLvl.bRtCompl = TRUE THEN
		tyP1080UsrMgmt.tyUsrMgmt.tyDrpDnLvl.bRtCompl	:= FALSE;
		bRefreshUsrMgmtTable 							:= TRUE;
	END_IF

	//Selected Row
	IF tyP1080Table.uiSelectedRow <> tyP1080Table.uiSelectedRowOld THEN
		FOR i := 1 TO c_uiP1080TableSize DO
			IF tyP1080Table.uiSelectedRow = i THEN
				tyP1080UsrMgmt.tyUsrMgmt.tyTableList.a_tyStringDataCol1[i].usiColor		:= 1;
				tyP1080UsrMgmt.tyUsrMgmt.tyTableList.a_tyTxtDataCol3[i].usiColor		:= 1;

			ELSE
				tyP1080UsrMgmt.tyUsrMgmt.tyTableList.a_tyStringDataCol1[i].usiColor		:= 0;
				tyP1080UsrMgmt.tyUsrMgmt.tyTableList.a_tyTxtDataCol3[i].usiColor		:= 0;

			END_IF
		END_FOR

		tyP1080Table.uiSelectedRowOld	:= tyP1080Table.uiSelectedRow;

	END_IF

	IF tyP1080UsrMgmt.tyUsrMgmt.tyTableList.a_tyStringDataCol1[tyP1080Table.uiSelectedRow].sValue = '' THEN
		fUIInRtStatOff(ADR(tyP1080UsrMgmt.tyUsrMgmt.tyBtnEditDetail.uiMaskRtStat));
		fUIInRtStatOff(ADR(tyP1080UsrMgmt.tyUsrMgmt.tyBtnDeleteUsr.uiMaskRtStat));
	ELSE
		fUIInRtStatHide(ADR(tyP1080UsrMgmt.tyUsrMgmt.tyBtnEditDetail.uiMaskRtStat));
		fUIInRtStatHide(ADR(tyP1080UsrMgmt.tyUsrMgmt.tyBtnDeleteUsr.uiMaskRtStat));
	END_IF

END_ACTION
```

#### Act_EntP1081Disp.st
```iecst
ACTION Act_EntP1081Disp:

	//Access Address
	p_tyC0004Navi ACCESS ADR(tyP1081UsrMgmtUsrAccessRgt.tyNaviBack);

	p_tyC0005Main ACCESS ADR(tyCommon.tyMain);

	p_tyC0006Set ACCESS ADR(tyCommon.tySet);

	p_tyC0007Notif ACCESS ADR(tyCommon.tyNotif);

	p_tyC0008MsgBox ACCESS ADR(tyP1081UsrMgmtUsrAccessRgt.tyMsgBoxHide);

	p_tyC0009Info ACCESS ADR(tyCommon.tyInfo);

	p_tyP1081UsrMgmtUsrAccessRgtSel ACCESS ADR(tyP1081UsrMgmtUsrAccessRgt.tyUsrAccessRgtSel);
	p_tyP1081UsrMgmtUsrAccessRgt ACCESS ADR(tyP1081UsrMgmtUsrAccessRgt.tyUsrAccessRgtLvl1);

	//Display
	//Reset Dropdown List
	tyP1081UsrMgmtUsrAccessRgt.tyUsrAccessRgtSel.tyDrpDnLevel.usiValueIdx	:= 0;

	//Backup Param
	tyP1081UsrMgmtUsrAccessRgt.tyUsrAccessRgtLvl1BkUp	:= tyP1081UsrMgmtUsrAccessRgt.tyUsrAccessRgtLvl1;
	tyP1081UsrMgmtUsrAccessRgt.tyUsrAccessRgtLvl2BkUp	:= tyP1081UsrMgmtUsrAccessRgt.tyUsrAccessRgtLvl2;
	tyP1081UsrMgmtUsrAccessRgt.tyUsrAccessRgtLvl3BkUp	:= tyP1081UsrMgmtUsrAccessRgt.tyUsrAccessRgtLvl3;

END_ACTION
```

#### Act_ExitP1081.st
```iecst
ACTION Act_ExitP1081:

	IF tyCommon.tySet.tyBtnSave.uiMaskRtStat.0 = FALSE THEN
		usiChgPage	:= 1;

	ELSE

		p_tyC0008MsgBox ACCESS ADR(tyP1081UsrMgmtUsrAccessRgt.tyMsgBoxExitAsk);

		IF tyP1081UsrMgmtUsrAccessRgt.tyMsgBoxExitAsk.tyBtnYes.bRtCompl = TRUE THEN
			tyP1081UsrMgmtUsrAccessRgt.tyMsgBoxExitAsk.tyBtnYes.bRtCompl	:= FALSE;
			tyP1081UsrMgmtUsrAccessRgt.tyMsgBoxExitAsk.tyBtnYes.bValue		:= FALSE;

			p_tyC0008MsgBox ACCESS ADR(tyP1081UsrMgmtUsrAccessRgt.tyMsgBoxHide);

			//Restore Param
			tyP1081UsrMgmtUsrAccessRgt.tyUsrAccessRgtLvl1	:= tyP1081UsrMgmtUsrAccessRgt.tyUsrAccessRgtLvl1BkUp;
			tyP1081UsrMgmtUsrAccessRgt.tyUsrAccessRgtLvl2	:= tyP1081UsrMgmtUsrAccessRgt.tyUsrAccessRgtLvl2BkUp;
			tyP1081UsrMgmtUsrAccessRgt.tyUsrAccessRgtLvl3	:= tyP1081UsrMgmtUsrAccessRgt.tyUsrAccessRgtLvl3BkUp;

			fUIInRtStatOff(ADR(tyCommon.tySet.tyBtnSave.uiMaskRtStat));

			usiChgPage	:= 1;

		ELSIF tyP1081UsrMgmtUsrAccessRgt.tyMsgBoxExitAsk.tyBtnNo.bRtCompl = TRUE THEN
			tyP1081UsrMgmtUsrAccessRgt.tyMsgBoxExitAsk.tyBtnNo.bRtCompl	:= FALSE;
			tyP1081UsrMgmtUsrAccessRgt.tyMsgBoxExitAsk.tyBtnNo.bValue	:= FALSE;

			p_tyC0008MsgBox ACCESS ADR(tyP1081UsrMgmtUsrAccessRgt.tyMsgBoxHide);

			eChgPage	:= eCurrPage;
			usiChgPage	:= 0;

		END_IF

	END_IF

END_ACTION
```

#### Act_OptP1081Navi.st
```iecst
ACTION Act_OptP1081Navi:

	tyP1081UsrMgmtUsrAccessRgt.tyNaviBack.tyBtnBack.bRtLk	:= tyCommon.tySet.tyBtnSave.bRtCompl;

	IF tyP1081UsrMgmtUsrAccessRgt.tyNaviBack.tyBtnBack.bRtCompl = TRUE THEN
		tyP1081UsrMgmtUsrAccessRgt.tyNaviBack.tyBtnBack.bRtCompl 	:= FALSE;
		tyP1081UsrMgmtUsrAccessRgt.tyNaviBack.tyBtnBack.bValue	 	:= FALSE;

		eChgPage	:= UIP1080UsrMgmt;

	END_IF

END_ACTION
```

#### Act_OptP1081Load.st
```iecst
ACTION Act_OptP1081Load:

	IF tyP1081UsrMgmtUsrAccessRgt.tyUsrAccessRgtSel.tyDrpDnLevel.bRtCompl = TRUE THEN
		tyP1081UsrMgmtUsrAccessRgt.tyUsrAccessRgtSel.tyDrpDnLevel.bRtCompl		:= FALSE;

		CASE tyP1081UsrMgmtUsrAccessRgt.tyUsrAccessRgtSel.tyDrpDnLevel.usiValueIdx OF
			0:
				p_tyP1081UsrMgmtUsrAccessRgt ACCESS ADR(tyP1081UsrMgmtUsrAccessRgt.tyUsrAccessRgtLvl1);

				fUIInRtStatOff(ADR(tyP1081UsrMgmtUsrAccessRgt.tyUsrAccessRgtLvl1.tyLyr.uiRtStat));
				fUIInRtStatHide(ADR(tyP1081UsrMgmtUsrAccessRgt.tyUsrAccessRgtLvl2.tyLyr.uiRtStat));
				fUIInRtStatHide(ADR(tyP1081UsrMgmtUsrAccessRgt.tyUsrAccessRgtLvl3.tyLyr.uiRtStat));

			1:
				p_tyP1081UsrMgmtUsrAccessRgt ACCESS ADR(tyP1081UsrMgmtUsrAccessRgt.tyUsrAccessRgtLvl2);

				fUIInRtStatHide(ADR(tyP1081UsrMgmtUsrAccessRgt.tyUsrAccessRgtLvl1.tyLyr.uiRtStat));
				fUIInRtStatOff(ADR(tyP1081UsrMgmtUsrAccessRgt.tyUsrAccessRgtLvl2.tyLyr.uiRtStat));
				fUIInRtStatHide(ADR(tyP1081UsrMgmtUsrAccessRgt.tyUsrAccessRgtLvl3.tyLyr.uiRtStat));

			2:
				p_tyP1081UsrMgmtUsrAccessRgt ACCESS ADR(tyP1081UsrMgmtUsrAccessRgt.tyUsrAccessRgtLvl3);

				fUIInRtStatHide(ADR(tyP1081UsrMgmtUsrAccessRgt.tyUsrAccessRgtLvl1.tyLyr.uiRtStat));
				fUIInRtStatHide(ADR(tyP1081UsrMgmtUsrAccessRgt.tyUsrAccessRgtLvl2.tyLyr.uiRtStat));
				fUIInRtStatOff(ADR(tyP1081UsrMgmtUsrAccessRgt.tyUsrAccessRgtLvl3.tyLyr.uiRtStat));

		END_CASE
	END_IF

END_ACTION
```

#### Act_OptP1081Save.st
```iecst
ACTION Act_OptP1081Save:

	// Level 1
	IF tyP1081UsrMgmtUsrAccessRgt.tyUsrAccessRgtLvl1.tyStringNm.bRtCompl 					OR tyP1081UsrMgmtUsrAccessRgt.tyUsrAccessRgtLvl1.tyBtnOps.bRtCompl
		OR tyP1081UsrMgmtUsrAccessRgt.tyUsrAccessRgtLvl1.tyBtnProdSel.bRtCompl				OR tyP1081UsrMgmtUsrAccessRgt.tyUsrAccessRgtLvl1.tyBtnMagSel.bRtCompl
		OR tyP1081UsrMgmtUsrAccessRgt.tyUsrAccessRgtLvl1.tyBtnMcInfo.bRtCompl				OR tyP1081UsrMgmtUsrAccessRgt.tyUsrAccessRgtLvl1.tyBtnAlm.bRtCompl
		OR tyP1081UsrMgmtUsrAccessRgt.tyUsrAccessRgtLvl1.tyBtnBffrInfo.bRtCompl				OR tyP1081UsrMgmtUsrAccessRgt.tyUsrAccessRgtLvl1.tyBtnOvenInfo.bRtCompl
		OR tyP1081UsrMgmtUsrAccessRgt.tyUsrAccessRgtLvl1.tyBtnMagInfo.bRtCompl				OR tyP1081UsrMgmtUsrAccessRgt.tyUsrAccessRgtLvl1.tyBtnLFCtrl.bRtCompl
		OR tyP1081UsrMgmtUsrAccessRgt.tyUsrAccessRgtLvl1.tyBtnManual.bRtCompl				OR tyP1081UsrMgmtUsrAccessRgt.tyUsrAccessRgtLvl1.tyBtnSimu.bRtCompl
		OR tyP1081UsrMgmtUsrAccessRgt.tyUsrAccessRgtLvl1.tyBtnProdSet.bRtCompl				OR tyP1081UsrMgmtUsrAccessRgt.tyUsrAccessRgtLvl1.tyBtnMagSet.bRtCompl
		OR tyP1081UsrMgmtUsrAccessRgt.tyUsrAccessRgtLvl1.tyBtnMcSet.bRtCompl				OR tyP1081UsrMgmtUsrAccessRgt.tyUsrAccessRgtLvl1.tyBtnLang.bRtCompl
		OR tyP1081UsrMgmtUsrAccessRgt.tyUsrAccessRgtLvl1.tyBtnLFSet.bRtCompl				OR tyP1081UsrMgmtUsrAccessRgt.tyUsrAccessRgtLvl1.tyBtnChgParam.bRtCompl

		// Level 2
		OR tyP1081UsrMgmtUsrAccessRgt.tyUsrAccessRgtLvl2.tyStringNm.bRtCompl 				OR tyP1081UsrMgmtUsrAccessRgt.tyUsrAccessRgtLvl2.tyBtnOps.bRtCompl
		OR tyP1081UsrMgmtUsrAccessRgt.tyUsrAccessRgtLvl2.tyBtnProdSel.bRtCompl				OR tyP1081UsrMgmtUsrAccessRgt.tyUsrAccessRgtLvl2.tyBtnMagSel.bRtCompl
		OR tyP1081UsrMgmtUsrAccessRgt.tyUsrAccessRgtLvl2.tyBtnMcInfo.bRtCompl				OR tyP1081UsrMgmtUsrAccessRgt.tyUsrAccessRgtLvl2.tyBtnAlm.bRtCompl
		OR tyP1081UsrMgmtUsrAccessRgt.tyUsrAccessRgtLvl2.tyBtnBffrInfo.bRtCompl				OR tyP1081UsrMgmtUsrAccessRgt.tyUsrAccessRgtLvl2.tyBtnOvenInfo.bRtCompl
		OR tyP1081UsrMgmtUsrAccessRgt.tyUsrAccessRgtLvl2.tyBtnMagInfo.bRtCompl				OR tyP1081UsrMgmtUsrAccessRgt.tyUsrAccessRgtLvl2.tyBtnLFCtrl.bRtCompl
		OR tyP1081UsrMgmtUsrAccessRgt.tyUsrAccessRgtLvl2.tyBtnManual.bRtCompl				OR tyP1081UsrMgmtUsrAccessRgt.tyUsrAccessRgtLvl2.tyBtnSimu.bRtCompl
		OR tyP1081UsrMgmtUsrAccessRgt.tyUsrAccessRgtLvl2.tyBtnProdSet.bRtCompl				OR tyP1081UsrMgmtUsrAccessRgt.tyUsrAccessRgtLvl2.tyBtnMagSet.bRtCompl
		OR tyP1081UsrMgmtUsrAccessRgt.tyUsrAccessRgtLvl2.tyBtnMcSet.bRtCompl				OR tyP1081UsrMgmtUsrAccessRgt.tyUsrAccessRgtLvl2.tyBtnLang.bRtCompl
		OR tyP1081UsrMgmtUsrAccessRgt.tyUsrAccessRgtLvl2.tyBtnLFSet.bRtCompl				OR tyP1081UsrMgmtUsrAccessRgt.tyUsrAccessRgtLvl2.tyBtnChgParam.bRtCompl

		// Level 3
		OR tyP1081UsrMgmtUsrAccessRgt.tyUsrAccessRgtLvl3.tyStringNm.bRtCompl 				OR tyP1081UsrMgmtUsrAccessRgt.tyUsrAccessRgtLvl3.tyBtnOps.bRtCompl
		OR tyP1081UsrMgmtUsrAccessRgt.tyUsrAccessRgtLvl3.tyBtnProdSel.bRtCompl				OR tyP1081UsrMgmtUsrAccessRgt.tyUsrAccessRgtLvl3.tyBtnMagSel.bRtCompl
		OR tyP1081UsrMgmtUsrAccessRgt.tyUsrAccessRgtLvl3.tyBtnMcInfo.bRtCompl				OR tyP1081UsrMgmtUsrAccessRgt.tyUsrAccessRgtLvl3.tyBtnAlm.bRtCompl
		OR tyP1081UsrMgmtUsrAccessRgt.tyUsrAccessRgtLvl3.tyBtnBffrInfo.bRtCompl				OR tyP1081UsrMgmtUsrAccessRgt.tyUsrAccessRgtLvl3.tyBtnOvenInfo.bRtCompl
		OR tyP1081UsrMgmtUsrAccessRgt.tyUsrAccessRgtLvl3.tyBtnMagInfo.bRtCompl				OR tyP1081UsrMgmtUsrAccessRgt.tyUsrAccessRgtLvl3.tyBtnLFCtrl.bRtCompl
		OR tyP1081UsrMgmtUsrAccessRgt.tyUsrAccessRgtLvl3.tyBtnManual.bRtCompl				OR tyP1081UsrMgmtUsrAccessRgt.tyUsrAccessRgtLvl3.tyBtnSimu.bRtCompl
		OR tyP1081UsrMgmtUsrAccessRgt.tyUsrAccessRgtLvl3.tyBtnProdSet.bRtCompl				OR tyP1081UsrMgmtUsrAccessRgt.tyUsrAccessRgtLvl3.tyBtnMagSet.bRtCompl
		OR tyP1081UsrMgmtUsrAccessRgt.tyUsrAccessRgtLvl3.tyBtnMcSet.bRtCompl				OR tyP1081UsrMgmtUsrAccessRgt.tyUsrAccessRgtLvl3.tyBtnLang.bRtCompl
		OR tyP1081UsrMgmtUsrAccessRgt.tyUsrAccessRgtLvl3.tyBtnLFSet.bRtCompl				OR tyP1081UsrMgmtUsrAccessRgt.tyUsrAccessRgtLvl3.tyBtnChgParam.bRtCompl				THEN

		fUIInRtStatHide(ADR(tyCommon.tySet.tyBtnSave.uiMaskRtStat));

		// Level 1
		tyP1081UsrMgmtUsrAccessRgt.tyUsrAccessRgtLvl1.tyStringNm.bRtCompl 		:= FALSE;
		tyP1081UsrMgmtUsrAccessRgt.tyUsrAccessRgtLvl1.tyBtnOps.bRtCompl 		:= FALSE;
		tyP1081UsrMgmtUsrAccessRgt.tyUsrAccessRgtLvl1.tyBtnProdSel.bRtCompl 	:= FALSE;
		tyP1081UsrMgmtUsrAccessRgt.tyUsrAccessRgtLvl1.tyBtnMagSel.bRtCompl 		:= FALSE;
		tyP1081UsrMgmtUsrAccessRgt.tyUsrAccessRgtLvl1.tyBtnMcInfo.bRtCompl		:= FALSE;
		tyP1081UsrMgmtUsrAccessRgt.tyUsrAccessRgtLvl1.tyBtnAlm.bRtCompl			:= FALSE;
		tyP1081UsrMgmtUsrAccessRgt.tyUsrAccessRgtLvl1.tyBtnBffrInfo.bRtCompl	:= FALSE;
		tyP1081UsrMgmtUsrAccessRgt.tyUsrAccessRgtLvl1.tyBtnOvenInfo.bRtCompl	:= FALSE;
		tyP1081UsrMgmtUsrAccessRgt.tyUsrAccessRgtLvl1.tyBtnMagInfo.bRtCompl		:= FALSE;
		tyP1081UsrMgmtUsrAccessRgt.tyUsrAccessRgtLvl1.tyBtnLFCtrl.bRtCompl		:= FALSE;
		tyP1081UsrMgmtUsrAccessRgt.tyUsrAccessRgtLvl1.tyBtnManual.bRtCompl		:= FALSE;
		tyP1081UsrMgmtUsrAccessRgt.tyUsrAccessRgtLvl1.tyBtnSimu.bRtCompl		:= FALSE;
		tyP1081UsrMgmtUsrAccessRgt.tyUsrAccessRgtLvl1.tyBtnProdSet.bRtCompl		:= FALSE;
		tyP1081UsrMgmtUsrAccessRgt.tyUsrAccessRgtLvl1.tyBtnMagSet.bRtCompl		:= FALSE;
		tyP1081UsrMgmtUsrAccessRgt.tyUsrAccessRgtLvl1.tyBtnMcSet.bRtCompl		:= FALSE;
		tyP1081UsrMgmtUsrAccessRgt.tyUsrAccessRgtLvl1.tyBtnLang.bRtCompl		:= FALSE;
		tyP1081UsrMgmtUsrAccessRgt.tyUsrAccessRgtLvl1.tyBtnLFSet.bRtCompl		:= FALSE;
		tyP1081UsrMgmtUsrAccessRgt.tyUsrAccessRgtLvl1.tyBtnChgParam.bRtCompl	:= FALSE;

		// Level 2
		tyP1081UsrMgmtUsrAccessRgt.tyUsrAccessRgtLvl2.tyStringNm.bRtCompl 		:= FALSE;
		tyP1081UsrMgmtUsrAccessRgt.tyUsrAccessRgtLvl2.tyBtnOps.bRtCompl 		:= FALSE;
		tyP1081UsrMgmtUsrAccessRgt.tyUsrAccessRgtLvl2.tyBtnProdSel.bRtCompl 	:= FALSE;
		tyP1081UsrMgmtUsrAccessRgt.tyUsrAccessRgtLvl2.tyBtnMagSel.bRtCompl 		:= FALSE;
		tyP1081UsrMgmtUsrAccessRgt.tyUsrAccessRgtLvl2.tyBtnMcInfo.bRtCompl		:= FALSE;
		tyP1081UsrMgmtUsrAccessRgt.tyUsrAccessRgtLvl2.tyBtnAlm.bRtCompl			:= FALSE;
		tyP1081UsrMgmtUsrAccessRgt.tyUsrAccessRgtLvl2.tyBtnBffrInfo.bRtCompl	:= FALSE;
		tyP1081UsrMgmtUsrAccessRgt.tyUsrAccessRgtLvl2.tyBtnOvenInfo.bRtCompl	:= FALSE;
		tyP1081UsrMgmtUsrAccessRgt.tyUsrAccessRgtLvl2.tyBtnMagInfo.bRtCompl		:= FALSE;
		tyP1081UsrMgmtUsrAccessRgt.tyUsrAccessRgtLvl2.tyBtnLFCtrl.bRtCompl		:= FALSE;
		tyP1081UsrMgmtUsrAccessRgt.tyUsrAccessRgtLvl2.tyBtnManual.bRtCompl		:= FALSE;
		tyP1081UsrMgmtUsrAccessRgt.tyUsrAccessRgtLvl2.tyBtnSimu.bRtCompl		:= FALSE;
		tyP1081UsrMgmtUsrAccessRgt.tyUsrAccessRgtLvl2.tyBtnProdSet.bRtCompl		:= FALSE;
		tyP1081UsrMgmtUsrAccessRgt.tyUsrAccessRgtLvl2.tyBtnMagSet.bRtCompl		:= FALSE;
		tyP1081UsrMgmtUsrAccessRgt.tyUsrAccessRgtLvl2.tyBtnMcSet.bRtCompl		:= FALSE;
		tyP1081UsrMgmtUsrAccessRgt.tyUsrAccessRgtLvl2.tyBtnLang.bRtCompl		:= FALSE;
		tyP1081UsrMgmtUsrAccessRgt.tyUsrAccessRgtLvl2.tyBtnLFSet.bRtCompl		:= FALSE;
		tyP1081UsrMgmtUsrAccessRgt.tyUsrAccessRgtLvl2.tyBtnChgParam.bRtCompl	:= FALSE;

		// Level 3
		tyP1081UsrMgmtUsrAccessRgt.tyUsrAccessRgtLvl3.tyStringNm.bRtCompl 		:= FALSE;
		tyP1081UsrMgmtUsrAccessRgt.tyUsrAccessRgtLvl3.tyBtnOps.bRtCompl 		:= FALSE;
		tyP1081UsrMgmtUsrAccessRgt.tyUsrAccessRgtLvl3.tyBtnProdSel.bRtCompl 	:= FALSE;
		tyP1081UsrMgmtUsrAccessRgt.tyUsrAccessRgtLvl3.tyBtnMagSel.bRtCompl 		:= FALSE;
		tyP1081UsrMgmtUsrAccessRgt.tyUsrAccessRgtLvl3.tyBtnMcInfo.bRtCompl		:= FALSE;
		tyP1081UsrMgmtUsrAccessRgt.tyUsrAccessRgtLvl3.tyBtnAlm.bRtCompl			:= FALSE;
		tyP1081UsrMgmtUsrAccessRgt.tyUsrAccessRgtLvl3.tyBtnBffrInfo.bRtCompl	:= FALSE;
		tyP1081UsrMgmtUsrAccessRgt.tyUsrAccessRgtLvl3.tyBtnOvenInfo.bRtCompl	:= FALSE;
		tyP1081UsrMgmtUsrAccessRgt.tyUsrAccessRgtLvl3.tyBtnMagInfo.bRtCompl		:= FALSE;
		tyP1081UsrMgmtUsrAccessRgt.tyUsrAccessRgtLvl3.tyBtnLFCtrl.bRtCompl		:= FALSE;
		tyP1081UsrMgmtUsrAccessRgt.tyUsrAccessRgtLvl3.tyBtnManual.bRtCompl		:= FALSE;
		tyP1081UsrMgmtUsrAccessRgt.tyUsrAccessRgtLvl3.tyBtnSimu.bRtCompl		:= FALSE;
		tyP1081UsrMgmtUsrAccessRgt.tyUsrAccessRgtLvl3.tyBtnProdSet.bRtCompl		:= FALSE;
		tyP1081UsrMgmtUsrAccessRgt.tyUsrAccessRgtLvl3.tyBtnMagSet.bRtCompl		:= FALSE;
		tyP1081UsrMgmtUsrAccessRgt.tyUsrAccessRgtLvl3.tyBtnMcSet.bRtCompl		:= FALSE;
		tyP1081UsrMgmtUsrAccessRgt.tyUsrAccessRgtLvl3.tyBtnLang.bRtCompl		:= FALSE;
		tyP1081UsrMgmtUsrAccessRgt.tyUsrAccessRgtLvl3.tyBtnLFSet.bRtCompl		:= FALSE;
		tyP1081UsrMgmtUsrAccessRgt.tyUsrAccessRgtLvl3.tyBtnChgParam.bRtCompl	:= FALSE;

	END_IF

	IF tyCommon.tySet.tyBtnSave.bRtCompl = TRUE THEN
		//Save Param
		CASE tyP1081UsrMgmtUsrAccessRgt.tyUsrAccessRgtSel.tyDrpDnLevel.usiValueIdx OF
			0:
				tyUsrMgmtAccessRightLvl1Wr.sNm					:= tyP1081UsrMgmtUsrAccessRgt.tyUsrAccessRgtLvl1.tyStringNm.sValue;
				tyUsrMgmtAccessRightLvl1Wr.bOpt					:= tyP1081UsrMgmtUsrAccessRgt.tyUsrAccessRgtLvl1.tyBtnOps.bValue;
				tyUsrMgmtAccessRightLvl1Wr.bProdSel				:= tyP1081UsrMgmtUsrAccessRgt.tyUsrAccessRgtLvl1.tyBtnProdSel.bValue;
				tyUsrMgmtAccessRightLvl1Wr.bMagSel				:= tyP1081UsrMgmtUsrAccessRgt.tyUsrAccessRgtLvl1.tyBtnMagSel.bValue;
				tyUsrMgmtAccessRightLvl1Wr.bMcInfo				:= tyP1081UsrMgmtUsrAccessRgt.tyUsrAccessRgtLvl1.tyBtnMcInfo.bValue;
				tyUsrMgmtAccessRightLvl1Wr.bAlm					:= tyP1081UsrMgmtUsrAccessRgt.tyUsrAccessRgtLvl1.tyBtnAlm.bValue;
				tyUsrMgmtAccessRightLvl1Wr.bBffrInfo			:= tyP1081UsrMgmtUsrAccessRgt.tyUsrAccessRgtLvl1.tyBtnBffrInfo.bValue;
				tyUsrMgmtAccessRightLvl1Wr.bOvenInfo			:= tyP1081UsrMgmtUsrAccessRgt.tyUsrAccessRgtLvl1.tyBtnOvenInfo.bValue;
				tyUsrMgmtAccessRightLvl1Wr.bMagInfo				:= tyP1081UsrMgmtUsrAccessRgt.tyUsrAccessRgtLvl1.tyBtnMagInfo.bValue;
				tyUsrMgmtAccessRightLvl1Wr.bLFCtrl				:= tyP1081UsrMgmtUsrAccessRgt.tyUsrAccessRgtLvl1.tyBtnLFCtrl.bValue;
				tyUsrMgmtAccessRightLvl1Wr.bManual				:= tyP1081UsrMgmtUsrAccessRgt.tyUsrAccessRgtLvl1.tyBtnManual.bValue;
				tyUsrMgmtAccessRightLvl1Wr.bSimulation			:= tyP1081UsrMgmtUsrAccessRgt.tyUsrAccessRgtLvl1.tyBtnSimu.bValue;
				tyUsrMgmtAccessRightLvl1Wr.bProdSet				:= tyP1081UsrMgmtUsrAccessRgt.tyUsrAccessRgtLvl1.tyBtnProdSet.bValue;
				tyUsrMgmtAccessRightLvl1Wr.bMagSet				:= tyP1081UsrMgmtUsrAccessRgt.tyUsrAccessRgtLvl1.tyBtnMagSet.bValue;
				tyUsrMgmtAccessRightLvl1Wr.bMcSet				:= tyP1081UsrMgmtUsrAccessRgt.tyUsrAccessRgtLvl1.tyBtnMcSet.bValue;
				tyUsrMgmtAccessRightLvl1Wr.bLang				:= tyP1081UsrMgmtUsrAccessRgt.tyUsrAccessRgtLvl1.tyBtnLang.bValue;
				tyUsrMgmtAccessRightLvl1Wr.bLFSet				:= tyP1081UsrMgmtUsrAccessRgt.tyUsrAccessRgtLvl1.tyBtnLFSet.bValue;
				tyUsrMgmtAccessRightLvl1Wr.bChgParam			:= tyP1081UsrMgmtUsrAccessRgt.tyUsrAccessRgtLvl1.tyBtnChgParam.bValue;

			1:
				tyUsrMgmtAccessRightLvl2Wr.sNm					:= tyP1081UsrMgmtUsrAccessRgt.tyUsrAccessRgtLvl2.tyStringNm.sValue;
				tyUsrMgmtAccessRightLvl2Wr.bOpt					:= tyP1081UsrMgmtUsrAccessRgt.tyUsrAccessRgtLvl2.tyBtnOps.bValue;
				tyUsrMgmtAccessRightLvl2Wr.bProdSel				:= tyP1081UsrMgmtUsrAccessRgt.tyUsrAccessRgtLvl2.tyBtnProdSel.bValue;
				tyUsrMgmtAccessRightLvl2Wr.bMagSel				:= tyP1081UsrMgmtUsrAccessRgt.tyUsrAccessRgtLvl2.tyBtnMagSel.bValue;
				tyUsrMgmtAccessRightLvl2Wr.bMcInfo				:= tyP1081UsrMgmtUsrAccessRgt.tyUsrAccessRgtLvl2.tyBtnMcInfo.bValue;
				tyUsrMgmtAccessRightLvl2Wr.bAlm					:= tyP1081UsrMgmtUsrAccessRgt.tyUsrAccessRgtLvl2.tyBtnAlm.bValue;
				tyUsrMgmtAccessRightLvl2Wr.bBffrInfo			:= tyP1081UsrMgmtUsrAccessRgt.tyUsrAccessRgtLvl2.tyBtnBffrInfo.bValue;
				tyUsrMgmtAccessRightLvl2Wr.bOvenInfo			:= tyP1081UsrMgmtUsrAccessRgt.tyUsrAccessRgtLvl2.tyBtnOvenInfo.bValue;
				tyUsrMgmtAccessRightLvl2Wr.bMagInfo				:= tyP1081UsrMgmtUsrAccessRgt.tyUsrAccessRgtLvl2.tyBtnMagInfo.bValue;
				tyUsrMgmtAccessRightLvl2Wr.bLFCtrl				:= tyP1081UsrMgmtUsrAccessRgt.tyUsrAccessRgtLvl2.tyBtnLFCtrl.bValue;
				tyUsrMgmtAccessRightLvl2Wr.bManual				:= tyP1081UsrMgmtUsrAccessRgt.tyUsrAccessRgtLvl2.tyBtnManual.bValue;
				tyUsrMgmtAccessRightLvl2Wr.bSimulation			:= tyP1081UsrMgmtUsrAccessRgt.tyUsrAccessRgtLvl2.tyBtnSimu.bValue;
				tyUsrMgmtAccessRightLvl2Wr.bProdSet				:= tyP1081UsrMgmtUsrAccessRgt.tyUsrAccessRgtLvl2.tyBtnProdSet.bValue;
				tyUsrMgmtAccessRightLvl2Wr.bMagSet				:= tyP1081UsrMgmtUsrAccessRgt.tyUsrAccessRgtLvl2.tyBtnMagSet.bValue;
				tyUsrMgmtAccessRightLvl2Wr.bMcSet				:= tyP1081UsrMgmtUsrAccessRgt.tyUsrAccessRgtLvl2.tyBtnMcSet.bValue;
				tyUsrMgmtAccessRightLvl2Wr.bLang				:= tyP1081UsrMgmtUsrAccessRgt.tyUsrAccessRgtLvl2.tyBtnLang.bValue;
				tyUsrMgmtAccessRightLvl2Wr.bLFSet				:= tyP1081UsrMgmtUsrAccessRgt.tyUsrAccessRgtLvl2.tyBtnLFSet.bValue;
				tyUsrMgmtAccessRightLvl2Wr.bChgParam			:= tyP1081UsrMgmtUsrAccessRgt.tyUsrAccessRgtLvl2.tyBtnChgParam.bValue;

			2:
				tyUsrMgmtAccessRightLvl3Wr.sNm					:= tyP1081UsrMgmtUsrAccessRgt.tyUsrAccessRgtLvl3.tyStringNm.sValue;
				tyUsrMgmtAccessRightLvl3Wr.bOpt					:= tyP1081UsrMgmtUsrAccessRgt.tyUsrAccessRgtLvl3.tyBtnOps.bValue;
				tyUsrMgmtAccessRightLvl3Wr.bProdSel				:= tyP1081UsrMgmtUsrAccessRgt.tyUsrAccessRgtLvl3.tyBtnProdSel.bValue;
				tyUsrMgmtAccessRightLvl3Wr.bMagSel				:= tyP1081UsrMgmtUsrAccessRgt.tyUsrAccessRgtLvl3.tyBtnMagSel.bValue;
				tyUsrMgmtAccessRightLvl3Wr.bMcInfo				:= tyP1081UsrMgmtUsrAccessRgt.tyUsrAccessRgtLvl3.tyBtnMcInfo.bValue;
				tyUsrMgmtAccessRightLvl3Wr.bAlm					:= tyP1081UsrMgmtUsrAccessRgt.tyUsrAccessRgtLvl3.tyBtnAlm.bValue;
				tyUsrMgmtAccessRightLvl3Wr.bBffrInfo			:= tyP1081UsrMgmtUsrAccessRgt.tyUsrAccessRgtLvl3.tyBtnBffrInfo.bValue;
				tyUsrMgmtAccessRightLvl3Wr.bOvenInfo			:= tyP1081UsrMgmtUsrAccessRgt.tyUsrAccessRgtLvl3.tyBtnOvenInfo.bValue;
				tyUsrMgmtAccessRightLvl3Wr.bMagInfo				:= tyP1081UsrMgmtUsrAccessRgt.tyUsrAccessRgtLvl3.tyBtnMagInfo.bValue;
				tyUsrMgmtAccessRightLvl3Wr.bLFCtrl				:= tyP1081UsrMgmtUsrAccessRgt.tyUsrAccessRgtLvl3.tyBtnLFCtrl.bValue;
				tyUsrMgmtAccessRightLvl3Wr.bManual				:= tyP1081UsrMgmtUsrAccessRgt.tyUsrAccessRgtLvl3.tyBtnManual.bValue;
				tyUsrMgmtAccessRightLvl3Wr.bSimulation			:= tyP1081UsrMgmtUsrAccessRgt.tyUsrAccessRgtLvl3.tyBtnSimu.bValue;
				tyUsrMgmtAccessRightLvl3Wr.bProdSet				:= tyP1081UsrMgmtUsrAccessRgt.tyUsrAccessRgtLvl3.tyBtnProdSet.bValue;
				tyUsrMgmtAccessRightLvl3Wr.bMagSet				:= tyP1081UsrMgmtUsrAccessRgt.tyUsrAccessRgtLvl3.tyBtnMagSet.bValue;
				tyUsrMgmtAccessRightLvl3Wr.bMcSet				:= tyP1081UsrMgmtUsrAccessRgt.tyUsrAccessRgtLvl3.tyBtnMcSet.bValue;
				tyUsrMgmtAccessRightLvl3Wr.bLang				:= tyP1081UsrMgmtUsrAccessRgt.tyUsrAccessRgtLvl3.tyBtnLang.bValue;
				tyUsrMgmtAccessRightLvl3Wr.bLFSet				:= tyP1081UsrMgmtUsrAccessRgt.tyUsrAccessRgtLvl3.tyBtnLFSet.bValue;
				tyUsrMgmtAccessRightLvl3Wr.bChgParam			:= tyP1081UsrMgmtUsrAccessRgt.tyUsrAccessRgtLvl3.tyBtnChgParam.bValue;
		END_CASE

		eUsrMgmtAct	:= UsrMgmtActSaveAccessRight;

		IF p_eUsrMgmtStat = UsrMgmtActSaveAccessRight AND p_eUsrMgmtStatus = Done THEN
			eUsrMgmtAct	:= UsrMgmtActIdle;

			//Backup Param
			tyP1081UsrMgmtUsrAccessRgt.tyUsrAccessRgtLvl1BkUp		:= tyP1081UsrMgmtUsrAccessRgt.tyUsrAccessRgtLvl1;
			tyP1081UsrMgmtUsrAccessRgt.tyUsrAccessRgtLvl2BkUp		:= tyP1081UsrMgmtUsrAccessRgt.tyUsrAccessRgtLvl2;
			tyP1081UsrMgmtUsrAccessRgt.tyUsrAccessRgtLvl3BkUp		:= tyP1081UsrMgmtUsrAccessRgt.tyUsrAccessRgtLvl3;

			CASE tyP1081UsrMgmtUsrAccessRgt.tyUsrAccessRgtSel.tyDrpDnLevel.usiValueIdx OF
				0:
					tyProperty.tyUITxtSnippets.sUsrMgmtUsrLv1Nm		:= tyP1081UsrMgmtUsrAccessRgt.tyUsrAccessRgtLvl1.tyStringNm.sValue;
				1:
					tyProperty.tyUITxtSnippets.sUsrMgmtUsrLv2Nm		:= tyP1081UsrMgmtUsrAccessRgt.tyUsrAccessRgtLvl2.tyStringNm.sValue;
				2:
					tyProperty.tyUITxtSnippets.sUsrMgmtUsrLv3Nm		:= tyP1081UsrMgmtUsrAccessRgt.tyUsrAccessRgtLvl3.tyStringNm.sValue;
			END_CASE

			tyCommon.tySet.tyBtnSave.bRtCompl						:= FALSE;

			fUIInRtStatOff(ADR(tyCommon.tySet.tyBtnSave.uiMaskRtStat));

		ELSIF p_eUsrMgmtStatus = Error THEN
			p_tyC0008MsgBox ACCESS ADR(tyP1081UsrMgmtUsrAccessRgt.tyMsgBoxSaveErr);

			IF tyP1081UsrMgmtUsrAccessRgt.tyMsgBoxSaveErr.tyBtnNo.bRtCompl = TRUE THEN
				tyP1081UsrMgmtUsrAccessRgt.tyMsgBoxSaveErr.tyBtnNo.bRtCompl 				:= FALSE;
				tyP1081UsrMgmtUsrAccessRgt.tyMsgBoxSaveErr.tyBtnNo.bValue 					:= FALSE;

				p_tyC0008MsgBox ACCESS ADR(tyP1081UsrMgmtUsrAccessRgt.tyMsgBoxHide);

				//Recover Param
				tyUsrMgmtAccessRightLvl1Wr	:= p_tyUsrMgmtFullData.tyAccessRightLvl1;
				tyUsrMgmtAccessRightLvl2Wr	:= p_tyUsrMgmtFullData.tyAccessRightLvl2;
				tyUsrMgmtAccessRightLvl3Wr	:= p_tyUsrMgmtFullData.tyAccessRightLvl3;

				tyP1081UsrMgmtUsrAccessRgt.tyUsrAccessRgtLvl1		:= tyP1081UsrMgmtUsrAccessRgt.tyUsrAccessRgtLvl1BkUp;
				tyP1081UsrMgmtUsrAccessRgt.tyUsrAccessRgtLvl2		:= tyP1081UsrMgmtUsrAccessRgt.tyUsrAccessRgtLvl2BkUp;
				tyP1081UsrMgmtUsrAccessRgt.tyUsrAccessRgtLvl3		:= tyP1081UsrMgmtUsrAccessRgt.tyUsrAccessRgtLvl3BkUp;

				tyCommon.tySet.tyBtnSave.bRtCompl					:= FALSE;
				fUIInRtStatOff(ADR(tyCommon.tySet.tyBtnSave.uiMaskRtStat));
			END_IF
		END_IF
	END_IF

END_ACTION
```

#### Act_OptP1081Keypad.st
```iecst
ACTION Act_OptP1081Keypad:

	IF fUIOutRtStatTPIsOpen(ADR(tyP1081UsrMgmtUsrAccessRgt.tyUsrAccessRgtLvl1.tyStringNm.uiRtStat)) = TRUE THEN
		tyProperty.tyKeypad.tyStringTitle.sKeypadTitle		:= tyP1081UsrMgmtUsrAccessRgt.tyUsrAccessRgtLvl1.tyStringNm.sKeypadTitle;

	ELSIF fUIOutRtStatTPIsOpen(ADR(tyP1081UsrMgmtUsrAccessRgt.tyUsrAccessRgtLvl2.tyStringNm.uiRtStat)) = TRUE THEN
		tyProperty.tyKeypad.tyStringTitle.sKeypadTitle		:= tyP1081UsrMgmtUsrAccessRgt.tyUsrAccessRgtLvl2.tyStringNm.sKeypadTitle;

	ELSIF fUIOutRtStatTPIsOpen(ADR(tyP1081UsrMgmtUsrAccessRgt.tyUsrAccessRgtLvl3.tyStringNm.uiRtStat)) = TRUE THEN
		tyProperty.tyKeypad.tyStringTitle.sKeypadTitle		:= tyP1081UsrMgmtUsrAccessRgt.tyUsrAccessRgtLvl3.tyStringNm.sKeypadTitle;

	END_IF

END_ACTION
```

#### Act_EntP1027Disp.st
```iecst
ACTION Act_EntP1027Disp:

	//Access Address
	p_tyC0004Navi ACCESS ADR(tyP1027McSetOpCon.tyNaviBack);

	p_tyC0005Main ACCESS ADR(tyCommon.tyMain);

	p_tyC0006Set ACCESS ADR(tyCommon.tySet);

	p_tyC0007Notif ACCESS ADR(tyCommon.tyNotif);

	p_tyC0008MsgBox ACCESS ADR (tyP1027McSetOpCon.tyMsgBoxHide);

	p_tyC0009Info ACCESS ADR(tyCommon.tyInfo);

	p_tyP1027McSetOpCon ACCESS ADR(tyP1027McSetOpCon.tyParam);

	//Backup Param
	tyP1027McSetOpCon.tyParamBkUp	:= tyP1027McSetOpCon.tyParam;

END_ACTION
```

#### Act_ExitP1027.st
```iecst
ACTION Act_ExitP1027:

	IF tyCommon.tySet.tyBtnSave.uiMaskRtStat.0 = FALSE THEN
		usiChgPage	:= 1;

	ELSE

		p_tyC0008MsgBox ACCESS ADR(tyP1027McSetOpCon.tyMsgBoxExitAsk);

		IF tyP1027McSetOpCon.tyMsgBoxExitAsk.tyBtnYes.bRtCompl = TRUE THEN
			tyP1027McSetOpCon.tyMsgBoxExitAsk.tyBtnYes.bRtCompl	:= FALSE;
			tyP1027McSetOpCon.tyMsgBoxExitAsk.tyBtnYes.bValue		:= FALSE;

			p_tyC0008MsgBox ACCESS ADR(tyP1027McSetOpCon.tyMsgBoxHide);

			//Restore Param
			tyP1027McSetOpCon.tyParam	:= tyP1027McSetOpCon.tyParamBkUp;

			fUIInRtStatOff(ADR(tyCommon.tySet.tyBtnSave.uiMaskRtStat));

			usiChgPage	:= 1;

		ELSIF tyP1027McSetOpCon.tyMsgBoxExitAsk.tyBtnNo.bRtCompl = TRUE THEN
			tyP1027McSetOpCon.tyMsgBoxExitAsk.tyBtnNo.bRtCompl	:= FALSE;
			tyP1027McSetOpCon.tyMsgBoxExitAsk.tyBtnNo.bValue		:= FALSE;

			p_tyC0008MsgBox ACCESS ADR(tyP1027McSetOpCon.tyMsgBoxHide);

			eChgPage	:= eCurrPage;
			usiChgPage	:= 0;

		END_IF

	END_IF

END_ACTION
```

#### Act_OptP1027Navi.st
```iecst
ACTION Act_OptP1027Navi:

	tyP1027McSetOpCon.tyNaviBack.tyBtnBack.bRtLk	:= tyCommon.tySet.tyBtnSave.bRtCompl;

	IF tyP1027McSetOpCon.tyNaviBack.tyBtnBack.bRtCompl = TRUE THEN
		tyP1027McSetOpCon.tyNaviBack.tyBtnBack.bRtCompl	:= FALSE;

		eChgPage	:= UIP1020McSetNavi;

	END_IF

END_ACTION
```

#### Act_OptP1027Save.st
```iecst
ACTION Act_OptP1027Save:

	IF tyP1027McSetOpCon.tyParam.tyNumLineNo.bRtCompl OR tyP1027McSetOpCon.tyParam.tyNumStatNo.bRtCompl OR
		tyP1027McSetOpCon.tyParam.tyNumStatIdx.bRtCompl OR tyP1027McSetOpCon.tyParam.tyNumFuNo.bRtCompl OR
		tyP1027McSetOpCon.tyParam.tyNumWorkPos.bRtCompl OR tyP1027McSetOpCon.tyParam.tyNumToolPos.bRtCompl OR
		tyP1027McSetOpCon.tyParam.tyNumProcessNo.bRtCompl OR tyP1027McSetOpCon.tyParam.tyStringProcessNm.bRtCompl OR
		tyP1027McSetOpCon.tyParam.tyStringApplication.bRtCompl OR tyP1027McSetOpCon.tyParam.tyBtnOpConEn.bRtCompl OR
		tyP1027McSetOpCon.tyParam.tyStringOpConSvrIP.bRtCompl OR tyP1027McSetOpCon.tyParam.tyNumOpConSvrPort.bRtCompl THEN

		fUIInRtStatHide(ADR(tyCommon.tySet.tyBtnSave.uiMaskRtStat));

		tyP1027McSetOpCon.tyParam.tyNumLineNo.bRtCompl			:= FALSE;
		tyP1027McSetOpCon.tyParam.tyNumStatNo.bRtCompl			:= FALSE;
		tyP1027McSetOpCon.tyParam.tyNumStatIdx.bRtCompl			:= FALSE;
		tyP1027McSetOpCon.tyParam.tyNumFuNo.bRtCompl			:= FALSE;
		tyP1027McSetOpCon.tyParam.tyNumWorkPos.bRtCompl			:= FALSE;
		tyP1027McSetOpCon.tyParam.tyNumToolPos.bRtCompl			:= FALSE;
		tyP1027McSetOpCon.tyParam.tyNumProcessNo.bRtCompl		:= FALSE;
		tyP1027McSetOpCon.tyParam.tyStringProcessNm.bRtCompl	:= FALSE;
		tyP1027McSetOpCon.tyParam.tyStringApplication.bRtCompl	:= FALSE;
		tyP1027McSetOpCon.tyParam.tyBtnOpConEn.bRtCompl			:= FALSE;
		tyP1027McSetOpCon.tyParam.tyStringOpConSvrIP.bRtCompl	:= FALSE;
		tyP1027McSetOpCon.tyParam.tyNumOpConSvrPort.bRtCompl	:= FALSE;

	END_IF

	IF tyCommon.tySet.tyBtnSave.bRtCompl = TRUE THEN

		tyMcParamWr.tyOpConParam.uiLineNo			:=  DINT_TO_UINT (tyP1027McSetOpCon.tyParam.tyNumLineNo.diValue);
		tyMcParamWr.tyOpConParam.uiStatNo			:=  DINT_TO_UINT (tyP1027McSetOpCon.tyParam.tyNumStatNo.diValue);
		tyMcParamWr.tyOpConParam.uiStatIdx			:=  DINT_TO_UINT (tyP1027McSetOpCon.tyParam.tyNumStatIdx.diValue);
		tyMcParamWr.tyOpConParam.uiFuNo				:=  DINT_TO_UINT (tyP1027McSetOpCon.tyParam.tyNumFuNo.diValue);
		tyMcParamWr.tyOpConParam.uiWorkPos			:=  DINT_TO_UINT (tyP1027McSetOpCon.tyParam.tyNumWorkPos.diValue);
		tyMcParamWr.tyOpConParam.uiToolPos			:=  DINT_TO_UINT (tyP1027McSetOpCon.tyParam.tyNumToolPos.diValue);
		tyMcParamWr.tyOpConParam.uiProcessNo		:=  DINT_TO_UINT (tyP1027McSetOpCon.tyParam.tyNumProcessNo.diValue);
		tyMcParamWr.tyOpConParam.sProcessName			:=  tyP1027McSetOpCon.tyParam.tyStringProcessNm.sValue;
		tyMcParamWr.tyOpConParam.sApplication			:=  tyP1027McSetOpCon.tyParam.tyStringApplication.sValue;
		tyMcParamWr.bOpConEn				:=  tyP1027McSetOpCon.tyParam.tyBtnOpConEn.bValue;
		tyMcParamWr.sOpConIPAddr			:=  tyP1027McSetOpCon.tyParam.tyStringOpConSvrIP.sValue;
		tyMcParamWr.uiOpConSvrPort			:=  DINT_TO_UINT (tyP1027McSetOpCon.tyParam.tyNumOpConSvrPort.diValue);

		eMcParamAct	:= McParamActWrite;

		IF p_eMcParamStat = McParamActWrite AND p_eMcParamStatus = Done THEN

			eMcParamAct	:= McParamActIdle;

			//Update BackUp Param
			tyP1027McSetOpCon.tyParamBkUp	:= tyP1027McSetOpCon.tyParam;

			tyCommon.tySet.tyBtnSave.bRtCompl 	:= FALSE;
			fUIInRtStatOff(ADR(tyCommon.tySet.tyBtnSave.uiMaskRtStat));

		ELSIF p_eMcParamStatus = Error THEN
			p_tyC0008MsgBox ACCESS ADR(tyP1027McSetOpCon.tyMsgBoxSaveErr);

			IF tyP1027McSetOpCon.tyMsgBoxSaveErr.tyBtnNo.bRtCompl = TRUE THEN
				tyP1027McSetOpCon.tyMsgBoxSaveErr.tyBtnNo.bRtCompl	:= FALSE;
				tyP1027McSetOpCon.tyMsgBoxSaveErr.tyBtnNo.bValue		:= FALSE;

				p_tyC0008MsgBox ACCESS ADR(tyP1027McSetOpCon.tyMsgBoxHide);

				//Restore Param
				tyP1027McSetOpCon.tyParam	:= tyP1027McSetOpCon.tyParamBkUp;
				tyMcParamWr						:= p_tyMcParamCurr;

				tyCommon.tySet.tyBtnSave.bRtCompl 	:= FALSE;
				fUIInRtStatOff(ADR(tyCommon.tySet.tyBtnSave.uiMaskRtStat));
			END_IF

		END_IF

	END_IF

END_ACTION
```

#### Act_OptP1027Keypad.st
```iecst
ACTION Act_OptP1027Keypad:

//	IF fUIOutRtStatTPIsOpen(ADR(tyP1027McSetOpCon.tyScan.tyStringTopScanSvrIP.uiRtStat)) = TRUE THEN
//		tyProperty.tyKeypad.tyStringTitle.sKeypadTitle	:= tyP1027McSetOpCon.tyScan.tyStringTopScanSvrIP.sKeypadTitle;
//
//	ELSIF fUIOutRtStatTPIsOpen(ADR(tyP1027McSetOpCon.tyScan.tyNumTopScanSvrPort.uiRtStat)) = TRUE THEN
//		tyProperty.tyKeypad.tyStringTitle.sKeypadTitle	:= tyP1027McSetOpCon.tyScan.tyNumTopScanSvrPort.sKeypadTitle;
//
//	ELSIF fUIOutRtStatTPIsOpen(ADR(tyP1027McSetOpCon.tyScan.tyStringBtmScanSvrIP.uiRtStat)) = TRUE THEN
//		tyProperty.tyKeypad.tyStringTitle.sKeypadTitle	:= tyP1027McSetOpCon.tyScan.tyStringBtmScanSvrIP.sKeypadTitle;
//
//	ELSIF fUIOutRtStatTPIsOpen(ADR(tyP1027McSetOpCon.tyScan.tyNumBtmScanSvrPort.uiRtStat)) = TRUE THEN
//		tyProperty.tyKeypad.tyStringTitle.sKeypadTitle	:= tyP1027McSetOpCon.tyScan.tyNumBtmScanSvrPort.sKeypadTitle;
//
//	END_IF

END_ACTION
```
